LIN {X 0,Y 262.97,Z 575.386,A -85,B 0,C 180,E1 -19356.909,E2 -19356.909} C_VEL
LIN {X 0,Y 260.228,Z 588.208,A -85,B 0,C 180,E1 -19358.543,E2 -19358.543} C_VEL
LIN {X 0,Y 257.272,Z 600.423,A -85,B 0,C 180,E1 -19360.441,E2 -19360.441} C_VEL
LIN {X 0,Y 253.997,Z 612.742,A -85,B 0,C 180,E1 -19362.789,E2 -19362.789} C_VEL
LIN {X 0,Y 250.762,Z 624.067,A -85,B 0,C 180,E1 -19365.442,E2 -19365.442} C_VEL
LIN {X 0,Y 248,Z 633.546,A -85,B 0,C 180,E1 -19368.164,E2 -19368.164} C_VEL
LIN {X 0,Y 245.68,Z 641.534,A -85,B 0,C 180,E1 -19370.952,E2 -19370.952} C_VEL
LIN {X 0,Y 243.839,Z 648.227,A -85,B 0,C 180,E1 -19373.798,E2 -19373.798} C_VEL
LIN {X 0,Y 242.309,Z 653.952,A -85,B 0,C 180,E1 -19376.827,E2 -19376.827} C_VEL
LIN {X 0,Y 241.294,Z 658.236,A -85,B 0,C 180,E1 -19379.68,E2 -19379.68} C_VEL
LIN {X 0,Y 240.647,Z 661.145,A -85,B 0,C 180,E1 -19382.119,E2 -19382.119} C_VEL
LIN {X 0,Y 239.931,Z 664.333,A -85,B 0,C 180,E1 -19385.862,E2 -19385.862} C_VEL
LIN {X 0,Y 239.747,Z 665.513,A -85,B 0,C 180,E1 -19387.996,E2 -19387.996} C_VEL
LIN {X 0,Y 239.749,Z 666.237,A -85,B 0,C 180,E1 -19390.343,E2 -19390.343} C_VEL
LIN {X 0,Y 239.913,Z 666.406,A -85,B 0,C 180,E1 -19392.915,E2 -19392.915} C_VEL
LIN {X 0,Y 240.248,Z 665.992,A -85,B 0,C 180,E1 -19395.405,E2 -19395.405} C_VEL
LIN {X 0,Y 241.228,Z 664.102,A -85,B 0,C 180,E1 -19399.244,E2 -19399.244} C_VEL
LIN {X 0,Y 242.501,Z 661.254,A -85,B 0,C 180,E1 -19402.51,E2 -19402.51} C_VEL
LIN {X 0,Y 244.221,Z 657.411,A -85,B 0,C 180,E1 -19405.652,E2 -19405.652} C_VEL
LIN {X 0,Y 246.913,Z 651.612,A -85,B 0,C 180,E1 -19409.179,E2 -19409.179} C_VEL
LIN {X 0,Y 250.029,Z 644.776,A -85,B 0,C 180,E1 -19412.367,E2 -19412.367} C_VEL
LIN {X 0,Y 253.779,Z 636.355,A -85,B 0,C 180,E1 -19415.455,E2 -19415.455} C_VEL
LIN {X 0,Y 257.848,Z 626.845,A -85,B 0,C 180,E1 -19418.248,E2 -19418.248} C_VEL
LIN {X 0,Y 261.578,Z 617.491,A -85,B 0,C 180,E1 -19420.493,E2 -19420.493} C_VEL
LIN {X 0,Y 265.656,Z 606.455,A -85,B 0,C 180,E1 -19422.67,E2 -19422.67} C_VEL
LIN {X 0,Y 269.706,Z 594.368,A -85,B 0,C 180,E1 -19424.61,E2 -19424.61} C_VEL
LIN {X 0,Y 272.359,Z 585.531,A -85,B 0,C 180,E1 -19425.809,E2 -19425.809} C_VEL
LIN {X 0,Y 272.47,Z 583.373,A -85,B 0,C 180,E1 -19426.196,E2 -19426.196} C_VEL
LIN {X 0,Y 270.942,Z 574.805,A -85,B 0,C 180,E1 -19428.023,E2 -19428.023} C_VEL
LIN {X 0,Y 268.039,Z 563.986,A -85,B 0,C 180,E1 -19430.46,E2 -19430.46} C_VEL
LIN {X 0,Y 264.172,Z 554.325,A -85,B 0,C 180,E1 -19432.894,E2 -19432.894} C_VEL
LIN {X 0,Y 260.406,Z 546.743,A -85,B 0,C 180,E1 -19435.059,E2 -19435.059} C_VEL
LIN {X 0,Y 257.562,Z 542.282,A -85,B 0,C 180,E1 -19436.621,E2 -19436.621} C_VEL
LIN {X 0,Y 255.07,Z 538.329,A -85,B 0,C 180,E1 -19438.026,E2 -19438.026} C_VEL
LIN {X 0,Y 252.392,Z 534.455,A -85,B 0,C 180,E1 -19439.597,E2 -19439.597} C_VEL
LIN {X 0,Y 251.603,Z 532.992,A -85,B 0,C 180,E1 -19440.11,E2 -19440.11} C_VEL
LIN {X 0,Y 249.06,Z 530.463,A -85,B 0,C 180,E1 -19441.616,E2 -19441.616} C_VEL
LIN {X 0,Y 247.762,Z 528.054,A -85,B 0,C 180,E1 -19442.54,E2 -19442.54} C_VEL
LIN {X 0,Y 244.664,Z 526.005,A -85,B 0,C 180,E1 -19444.53,E2 -19444.53} C_VEL
LIN {X 0,Y 243.293,Z 523.765,A -85,B 0,C 180,E1 -19445.698,E2 -19445.698} C_VEL
LIN {X 0,Y 243.002,Z 522.69,A -85,B 0,C 180,E1 -19446.069,E2 -19446.069} C_VEL
LIN {X 0,Y 243.031,Z 522.727,A -85,B 0,C 180,E1 -19449.991,E2 -19449.991} C_VEL
LIN {X 0,Y 242.931,Z 523.303,A -85,B 0,C 180,E1 -19455.091,E2 -19455.091} C_VEL
LIN {X 0,Y 242.977,Z 524.161,A -85,B 0,C 180,E1 -19459.142,E2 -19459.142} C_VEL
LIN {X 0,Y 243.11,Z 525.075,A -85,B 0,C 180,E1 -19462.32,E2 -19462.32} C_VEL
LIN {X 0,Y 243.39,Z 526.569,A -85,B 0,C 180,E1 -19466.3,E2 -19466.3} C_VEL
LIN {X 0,Y 243.223,Z 527.205,A -85,B 0,C 180,E1 -19467.212,E2 -19467.212} C_VEL
LIN {X 0,Y 241.941,Z 529.538,A -85,B 0,C 180,E1 -19468.969,E2 -19468.969} C_VEL
LIN {X 0,Y 240.107,Z 534.806,A -85,B 0,C 180,E1 -19471.983,E2 -19471.983} C_VEL
LIN {X 0,Y 240.927,Z 536.647,A -85,B 0,C 180,E1 -19473.294,E2 -19473.294} C_VEL
LIN {X 0,Y 241.911,Z 537.613,A -85,B 0,C 180,E1 -19474.066,E2 -19474.066} C_VEL
LIN {X 0,Y 243.456,Z 541.241,A -85,B 0,C 180,E1 -19475.456,E2 -19475.456} C_VEL
LIN {X 0,Y 246.202,Z 544.885,A -85,B 0,C 180,E1 -19477.383,E2 -19477.383} C_VEL
LIN {X 0,Y 247.899,Z 548.7,A -85,B 0,C 180,E1 -19478.651,E2 -19478.651} C_VEL
LIN {X 0,Y 249.696,Z 551.295,A -85,B 0,C 180,E1 -19479.75,E2 -19479.75} C_VEL
LIN {X 0,Y 251.774,Z 555.814,A -85,B 0,C 180,E1 -19481.168,E2 -19481.168} C_VEL
LIN {X 0,Y 252.748,Z 557.67,A -85,B 0,C 180,E1 -19481.75,E2 -19481.75} C_VEL
LIN {X 0,Y 254.725,Z 561.939,A -85,B 0,C 180,E1 -19483.004,E2 -19483.004} C_VEL
LIN {X 0,Y 257.009,Z 569.051,A -85,B 0,C 180,E1 -19484.685,E2 -19484.685} C_VEL
LIN {X 0,Y 259.21,Z 578.738,A -85,B 0,C 180,E1 -19486.695,E2 -19486.695} C_VEL
LIN {X 0,Y 260.8,Z 588.921,A -85,B 0,C 180,E1 -19488.655,E2 -19488.655} C_VEL
LIN {X 0,Y 261.444,Z 600.468,A -85,B 0,C 180,E1 -19490.766,E2 -19490.766} C_VEL
LIN {X 0,Y 261.212,Z 611.698,A -85,B 0,C 180,E1 -19492.793,E2 -19492.793} C_VEL
LIN {X 0,Y 260.405,Z 619.56,A -85,B 0,C 180,E1 -19494.256,E2 -19494.256} C_VEL
LIN {X 0,Y 256.112,Z 631.595,A -85,B 0,C 180,E1 -19496.242,E2 -19496.242} C_VEL
LIN {X 0,Y 251.789,Z 642.638,A -85,B 0,C 180,E1 -19498.442,E2 -19498.442} C_VEL
LIN {X 0,Y 247.254,Z 653.496,A -85,B 0,C 180,E1 -19501.104,E2 -19501.104} C_VEL
LIN {X 0,Y 243.504,Z 662.394,A -85,B 0,C 180,E1 -19503.806,E2 -19503.806} C_VEL
LIN {X 0,Y 240.232,Z 670.29,A -85,B 0,C 180,E1 -19506.737,E2 -19506.737} C_VEL
LIN {X 0,Y 237.315,Z 677.59,A -85,B 0,C 180,E1 -19510.088,E2 -19510.088} C_VEL
LIN {X 0,Y 235.092,Z 683.518,A -85,B 0,C 180,E1 -19513.553,E2 -19513.553} C_VEL
LIN {X 0,Y 234.041,Z 687.003,A -85,B 0,C 180,E1 -19516.099,E2 -19516.099} C_VEL
LIN {X 0,Y 233.12,Z 690.607,A -85,B 0,C 180,E1 -19519.578,E2 -19519.578} C_VEL
LIN {X 0,Y 232.871,Z 693.033,A -85,B 0,C 180,E1 -19523.066,E2 -19523.066} C_VEL
LIN {X 0,Y 232.938,Z 694.303,A -85,B 0,C 180,E1 -19526.54,E2 -19526.54} C_VEL
LIN {X 0,Y 233.106,Z 694.406,A -85,B 0,C 180,E1 -19529.999,E2 -19529.999} C_VEL
LIN {X 0,Y 233.01,Z 693.243,A -85,B 0,C 180,E1 -19533.457,E2 -19533.457} C_VEL
LIN {X 0,Y 233.026,Z 691.945,A -85,B 0,C 180,E1 -19535.58,E2 -19535.58} C_VEL
LIN {X 0,Y 233.094,Z 688.21,A -85,B 0,C 180,E1 -19539.544,E2 -19539.544} C_VEL
LIN {X 0,Y 233.729,Z 683.513,A -85,B 0,C 180,E1 -19543.032,E2 -19543.032} C_VEL
LIN {X 0,Y 234.925,Z 677.626,A -85,B 0,C 180,E1 -19546.359,E2 -19546.359} C_VEL
LIN {X 0,Y 236.712,Z 670.612,A -85,B 0,C 180,E1 -19549.511,E2 -19549.511} C_VEL
LIN {X 0,Y 239.023,Z 662.501,A -85,B 0,C 180,E1 -19552.471,E2 -19552.471} C_VEL
LIN {X 0,Y 241.896,Z 652.756,A -85,B 0,C 180,E1 -19555.374,E2 -19555.374} C_VEL
LIN {X 0,Y 244.744,Z 642.794,A -85,B 0,C 180,E1 -19557.814,E2 -19557.814} C_VEL
LIN {X 0,Y 248.126,Z 631.005,A -85,B 0,C 180,E1 -19560.181,E2 -19560.181} C_VEL
LIN {X 0,Y 251.301,Z 619.334,A -85,B 0,C 180,E1 -19562.096,E2 -19562.096} C_VEL
LIN {X 0,Y 252.22,Z 615.752,A -85,B 0,C 180,E1 -19562.622,E2 -19562.622} C_VEL
LIN {X 0,Y 252.245,Z 609.63,A -85,B 0,C 180,E1 -19563.595,E2 -19563.595} C_VEL
LIN {X 0,Y 251.323,Z 597.034,A -85,B 0,C 180,E1 -19565.49,E2 -19565.49} C_VEL
LIN {X 0,Y 249.511,Z 583.538,A -85,B 0,C 180,E1 -19567.341,E2 -19567.341} C_VEL
LIN {X 0,Y 246.829,Z 569.413,A -85,B 0,C 180,E1 -19569.11,E2 -19569.11} C_VEL
LIN {X 0,Y 243.114,Z 554.934,A -85,B 0,C 180,E1 -19570.776,E2 -19570.776} C_VEL
LIN {X 0,Y 238.76,Z 541.769,A -85,B 0,C 180,E1 -19572.228,E2 -19572.228} C_VEL
LIN {X 0,Y 237.734,Z 538.235,A -85,B 0,C 180,E1 -19572.574,E2 -19572.574} C_VEL
LIN {X 0,Y 237.777,Z 535.861,A -85,B 0,C 180,E1 -19574.817,E2 -19574.817} C_VEL
LIN {X 0,Y 237.287,Z 532.906,A -85,B 0,C 180,E1 -19577.768,E2 -19577.768} C_VEL
LIN {X 0,Y 236.558,Z 529.52,A -85,B 0,C 180,E1 -19581.399,E2 -19581.399} C_VEL
LIN {X 0,Y 235.911,Z 525.797,A -85,B 0,C 180,E1 -19585.527,E2 -19585.527} C_VEL
LIN {X 0,Y 235.357,Z 522.081,A -85,B 0,C 180,E1 -19589.99,E2 -19589.99} C_VEL
LIN {X 0,Y 235.001,Z 519.837,A -85,B 0,C 180,E1 -19593.107,E2 -19593.107} C_VEL
LIN {X 0,Y 234.97,Z 519.844,A -85,B 0,C 180,E1 -19598,E2 -19598} C_VEL
LIN {X 0,Y 235.089,Z 519.827,A -85,B 0,C 180,E1 -19603.06,E2 -19603.06} C_VEL
LIN {X 0,Y 235.139,Z 519.815,A -85,B 0,C 180,E1 -19607.924,E2 -19607.924} C_VEL
LIN {X 0,Y 235.369,Z 519.771,A -85,B 0,C 180,E1 -19611.414,E2 -19611.414} C_VEL
LIN {X 0,Y 235.397,Z 519.778,A -85,B 0,C 180,E1 -19613.142,E2 -19613.142} C_VEL
LIN {X 0,Y 235.592,Z 519.755,A -85,B 0,C 180,E1 -19618.291,E2 -19618.291} C_VEL
LIN {X 0,Y 235.59,Z 519.741,A -85,B 0,C 180,E1 -19621.71,E2 -19621.71} C_VEL
LIN {X 0,Y 235.387,Z 519.788,A -85,B 0,C 180,E1 -19626.86,E2 -19626.86} C_VEL
LIN {X 0,Y 235.208,Z 519.795,A -85,B 0,C 180,E1 -19630.329,E2 -19630.329} C_VEL
LIN {X 0,Y 235.106,Z 519.816,A -85,B 0,C 180,E1 -19635.608,E2 -19635.608} C_VEL
LIN {X 0,Y 235.003,Z 519.837,A -85,B 0,C 180,E1 -19639.207,E2 -19639.207} C_VEL
LIN {X 0,Y 234.956,Z 519.819,A -85,B 0,C 180,E1 -19642.884,E2 -19642.884} C_VEL
LIN {X 0,Y 234.965,Z 519.83,A -85,B 0,C 180,E1 -19646.659,E2 -19646.659} C_VEL
LIN {X 0,Y 234.928,Z 519.844,A -85,B 0,C 180,E1 -19650.569,E2 -19650.569} C_VEL
LIN {X 0,Y 234.957,Z 519.821,A -85,B 0,C 180,E1 -19654.634,E2 -19654.634} C_VEL
LIN {X 0,Y 234.964,Z 519.835,A -85,B 0,C 180,E1 -19658.954,E2 -19658.954} C_VEL
LIN {X 0,Y 234.995,Z 519.832,A -85,B 0,C 180,E1 -19663.462,E2 -19663.462} C_VEL
LIN {X 0,Y 234.991,Z 519.817,A -85,B 0,C 180,E1 -19666.54,E2 -19666.54} C_VEL
LIN {X 0,Y 234.954,Z 519.846,A -85,B 0,C 180,E1 -19671.088,E2 -19671.088} C_VEL
LIN {X 0,Y 234.961,Z 519.828,A -85,B 0,C 180,E1 -19675.369,E2 -19675.369} C_VEL
LIN {X 0,Y 234.97,Z 519.844,A -85,B 0,C 180,E1 -19680.159,E2 -19680.159} C_VEL
LIN {X 0,Y 234.996,Z 519.826,A -85,B 0,C 180,E1 -19683.795,E2 -19683.795} C_VEL
LIN {X 0,Y 235.014,Z 519.831,A -85,B 0,C 180,E1 -19688.971,E2 -19688.971} C_VEL
LIN {X 0,Y 235.1,Z 519.825,A -85,B 0,C 180,E1 -19693.061,E2 -19693.061} C_VEL
LIN {X 0,Y 235.147,Z 519.821,A -85,B 0,C 180,E1 -19697.925,E2 -19697.925} C_VEL
LIN {X 0,Y 235.33,Z 519.792,A -85,B 0,C 180,E1 -19701.413,E2 -19701.413} C_VEL
LIN {X 0,Y 235.373,Z 519.791,A -85,B 0,C 180,E1 -19703.141,E2 -19703.141} C_VEL
LIN {X 0,Y 235.421,Z 519.781,A -85,B 0,C 180,E1 -19707.381,E2 -19707.381} C_VEL
LIN {X 0,Y 236.515,Z 522.659,A -85,B 0,C 180,E1 -19707.742,E2 -19707.742} C_VEL
LIN {X 0,Y 238.065,Z 524.891,A -85,B 0,C 180,E1 -19708.151,E2 -19708.151} C_VEL
LIN {X 0,Y 242.678,Z 533.731,A -85,B 0,C 180,E1 -19709.542,E2 -19709.542} C_VEL
LIN {X 0,Y 249.035,Z 548.124,A -85,B 0,C 180,E1 -19711.775,E2 -19711.775} C_VEL
LIN {X 0,Y 252.052,Z 557.462,A -85,B 0,C 180,E1 -19713.198,E2 -19713.198} C_VEL
LIN {X 0,Y 255.332,Z 570.437,A -85,B 0,C 180,E1 -19715.255,E2 -19715.255} C_VEL
LIN {X 0,Y 256.488,Z 576.766,A -85,B 0,C 180,E1 -19716.293,E2 -19716.293} C_VEL
LIN {X 0,Y 253.332,Z 590.847,A -85,B 0,C 180,E1 -19718.175,E2 -19718.175} C_VEL
LIN {X 0,Y 250.031,Z 603.805,A -85,B 0,C 180,E1 -19720.324,E2 -19720.324} C_VEL
LIN {X 0,Y 246.656,Z 615.754,A -85,B 0,C 180,E1 -19722.758,E2 -19722.758} C_VEL
LIN {X 0,Y 243.418,Z 626.66,A -85,B 0,C 180,E1 -19725.49,E2 -19725.49} C_VEL
LIN {X 0,Y 240.665,Z 635.779,A -85,B 0,C 180,E1 -19728.297,E2 -19728.297} C_VEL
LIN {X 0,Y 238.341,Z 643.461,A -85,B 0,C 180,E1 -19731.175,E2 -19731.175} C_VEL
LIN {X 0,Y 236.222,Z 650.859,A -85,B 0,C 180,E1 -19734.616,E2 -19734.616} C_VEL
LIN {X 0,Y 234.883,Z 655.996,A -85,B 0,C 180,E1 -19737.632,E2 -19737.632} C_VEL
LIN {X 0,Y 233.887,Z 660.153,A -85,B 0,C 180,E1 -19740.719,E2 -19740.719} C_VEL
LIN {X 0,Y 233.36,Z 662.351,A -85,B 0,C 180,E1 -19742.827,E2 -19742.827} C_VEL
LIN {X 0,Y 232.882,Z 664.441,A -85,B 0,C 180,E1 -19745.429,E2 -19745.429} C_VEL
LIN {X 0,Y 232.633,Z 666.379,A -85,B 0,C 180,E1 -19749.378,E2 -19749.378} C_VEL
LIN {X 0,Y 232.725,Z 666.833,A -85,B 0,C 180,E1 -19751.634,E2 -19751.634} C_VEL
LIN {X 0,Y 232.936,Z 666.819,A -85,B 0,C 180,E1 -19753.943,E2 -19753.943} C_VEL
LIN {X 0,Y 233.325,Z 666.251,A -85,B 0,C 180,E1 -19756.295,E2 -19756.295} C_VEL
LIN {X 0,Y 233.963,Z 665.147,A -85,B 0,C 180,E1 -19758.675,E2 -19758.675} C_VEL
LIN {X 0,Y 235.285,Z 662.487,A -85,B 0,C 180,E1 -19762.261,E2 -19762.261} C_VEL
LIN {X 0,Y 237.336,Z 658.263,A -85,B 0,C 180,E1 -19766.01,E2 -19766.01} C_VEL
LIN {X 0,Y 239.932,Z 653.095,A -85,B 0,C 180,E1 -19769.35,E2 -19769.35} C_VEL
LIN {X 0,Y 242.909,Z 647.003,A -85,B 0,C 180,E1 -19772.423,E2 -19772.423} C_VEL
LIN {X 0,Y 246.185,Z 640.109,A -85,B 0,C 180,E1 -19775.203,E2 -19775.203} C_VEL
LIN {X 0,Y 250.414,Z 630.965,A -85,B 0,C 180,E1 -19778.172,E2 -19778.172} C_VEL
LIN {X 0,Y 254.916,Z 620.513,A -85,B 0,C 180,E1 -19780.889,E2 -19780.889} C_VEL
LIN {X 0,Y 259.401,Z 609.166,A -85,B 0,C 180,E1 -19783.269,E2 -19783.269} C_VEL
LIN {X 0,Y 263.785,Z 596.954,A -85,B 0,C 180,E1 -19785.338,E2 -19785.338} C_VEL
LIN {X 0,Y 266.902,Z 587.098,A -85,B 0,C 180,E1 -19786.717,E2 -19786.717} C_VEL
LIN {X 0,Y 265.723,Z 578.921,A -85,B 0,C 180,E1 -19788.558,E2 -19788.558} C_VEL
LIN {X 0,Y 263.505,Z 569.481,A -85,B 0,C 180,E1 -19790.791,E2 -19790.791} C_VEL
LIN {X 0,Y 260.847,Z 561.758,A -85,B 0,C 180,E1 -19792.803,E2 -19792.803} C_VEL
LIN {X 0,Y 257.119,Z 553.218,A -85,B 0,C 180,E1 -19795.296,E2 -19795.296} C_VEL
LIN {X 0,Y 254.632,Z 548.771,A -85,B 0,C 180,E1 -19796.835,E2 -19796.835} C_VEL
LIN {X 0,Y 251.808,Z 544.068,A -85,B 0,C 180,E1 -19798.63,E2 -19798.63} C_VEL
LIN {X 0,Y 249.334,Z 540.251,A -85,B 0,C 180,E1 -19800.226,E2 -19800.226} C_VEL
LIN {X 0,Y 248.552,Z 539.039,A -85,B 0,C 180,E1 -19800.759,E2 -19800.759} C_VEL
LIN {X 0,Y 246.294,Z 536.366,A -85,B 0,C 180,E1 -19802.277,E2 -19802.277} C_VEL
LIN {X 0,Y 245.257,Z 534.562,A -85,B 0,C 180,E1 -19803.079,E2 -19803.079} C_VEL
LIN {X 0,Y 242.481,Z 532.36,A -85,B 0,C 180,E1 -19805.092,E2 -19805.092} C_VEL
LIN {X 0,Y 241.054,Z 529.742,A -85,B 0,C 180,E1 -19806.434,E2 -19806.434} C_VEL
LIN {X 0,Y 237.552,Z 527.249,A -85,B 0,C 180,E1 -19809.794,E2 -19809.794} C_VEL
LIN {X 0,Y 236.193,Z 525.11,A -85,B 0,C 180,E1 -19811.804,E2 -19811.804} C_VEL
LIN {X 0,Y 235.995,Z 524.537,A -85,B 0,C 180,E1 -19812.25,E2 -19812.25} C_VEL
LIN {X 0,Y 236.03,Z 524.997,A -85,B 0,C 180,E1 -19815.544,E2 -19815.544} C_VEL
LIN {X 0,Y 236.063,Z 525.768,A -85,B 0,C 180,E1 -19819.116,E2 -19819.116} C_VEL
LIN {X 0,Y 236.222,Z 526.838,A -85,B 0,C 180,E1 -19822.753,E2 -19822.753} C_VEL
LIN {X 0,Y 236.505,Z 528.439,A -85,B 0,C 180,E1 -19826.94,E2 -19826.94} C_VEL
LIN {X 0,Y 236.652,Z 529.379,A -85,B 0,C 180,E1 -19828.611,E2 -19828.611} C_VEL
LIN {X 0,Y 238.401,Z 533.574,A -85,B 0,C 180,E1 -19830.95,E2 -19830.95} C_VEL
LIN {X 0,Y 240.927,Z 536.647,A -85,B 0,C 180,E1 -19833.294,E2 -19833.294} C_VEL
LIN {X 0,Y 241.916,Z 538.055,A -85,B 0,C 180,E1 -19834.124,E2 -19834.124} C_VEL
LIN {X 0,Y 243.061,Z 541.33,A -85,B 0,C 180,E1 -19835.247,E2 -19835.247} C_VEL
LIN {X 0,Y 243.881,Z 545.39,A -85,B 0,C 180,E1 -19836.251,E2 -19836.251} C_VEL
LIN {X 0,Y 245.389,Z 554.106,A -85,B 0,C 180,E1 -19838.231,E2 -19838.231} C_VEL
LIN {X 0,Y 246.185,Z 556.608,A -85,B 0,C 180,E1 -19838.953,E2 -19838.953} C_VEL
LIN {X 0,Y 248.839,Z 562.367,A -85,B 0,C 180,E1 -19840.919,E2 -19840.919} C_VEL
LIN {X 0,Y 251.791,Z 570.132,A -85,B 0,C 180,E1 -19843.145,E2 -19843.145} C_VEL
LIN {X 0,Y 253.95,Z 580.016,A -85,B 0,C 180,E1 -19845.372,E2 -19845.372} C_VEL
LIN {X 0,Y 255.419,Z 590.889,A -85,B 0,C 180,E1 -19847.614,E2 -19847.614} C_VEL
LIN {X 0,Y 255.913,Z 601.984,A -85,B 0,C 180,E1 -19849.761,E2 -19849.761} C_VEL
LIN {X 0,Y 255.478,Z 612.786,A -85,B 0,C 180,E1 -19851.841,E2 -19851.841} C_VEL
LIN {X 0,Y 254.531,Z 620.794,A -85,B 0,C 180,E1 -19853.393,E2 -19853.393} C_VEL
LIN {X 0,Y 250.259,Z 632.18,A -85,B 0,C 180,E1 -19855.342,E2 -19855.342} C_VEL
LIN {X 0,Y 245.782,Z 643.009,A -85,B 0,C 180,E1 -19857.578,E2 -19857.578} C_VEL
LIN {X 0,Y 241.047,Z 653.694,A -85,B 0,C 180,E1 -19860.287,E2 -19860.287} C_VEL
LIN {X 0,Y 237.004,Z 662.754,A -85,B 0,C 180,E1 -19863.121,E2 -19863.121} C_VEL
LIN {X 0,Y 233.671,Z 670.313,A -85,B 0,C 180,E1 -19866.044,E2 -19866.044} C_VEL
LIN {X 0,Y 230.591,Z 677.488,A -85,B 0,C 180,E1 -19869.482,E2 -19869.482} C_VEL
LIN {X 0,Y 228.152,Z 683.517,A -85,B 0,C 180,E1 -19873.164,E2 -19873.164} C_VEL
LIN {X 0,Y 227.085,Z 686.778,A -85,B 0,C 180,E1 -19875.664,E2 -19875.664} C_VEL
LIN {X 0,Y 226.08,Z 690.314,A -85,B 0,C 180,E1 -19879.25,E2 -19879.25} C_VEL
LIN {X 0,Y 225.785,Z 692.672,A -85,B 0,C 180,E1 -19882.847,E2 -19882.847} C_VEL
LIN {X 0,Y 225.855,Z 693.883,A -85,B 0,C 180,E1 -19886.431,E2 -19886.431} C_VEL
LIN {X 0,Y 226.027,Z 693.927,A -85,B 0,C 180,E1 -19889.999,E2 -19889.999} C_VEL
LIN {X 0,Y 225.924,Z 692.734,A -85,B 0,C 180,E1 -19893.566,E2 -19893.566} C_VEL
LIN {X 0,Y 225.955,Z 691.531,A -85,B 0,C 180,E1 -19895.554,E2 -19895.554} C_VEL
LIN {X 0,Y 225.948,Z 688.536,A -85,B 0,C 180,E1 -19898.946,E2 -19898.946} C_VEL
LIN {X 0,Y 226.476,Z 684.098,A -85,B 0,C 180,E1 -19902.545,E2 -19902.545} C_VEL
LIN {X 0,Y 227.696,Z 678.236,A -85,B 0,C 180,E1 -19906.127,E2 -19906.127} C_VEL
LIN {X 0,Y 229.626,Z 670.797,A -85,B 0,C 180,E1 -19909.673,E2 -19909.673} C_VEL
LIN {X 0,Y 231.999,Z 662.821,A -85,B 0,C 180,E1 -19912.719,E2 -19912.719} C_VEL
LIN {X 0,Y 234.956,Z 653.23,A -85,B 0,C 180,E1 -19915.703,E2 -19915.703} C_VEL
LIN {X 0,Y 237.827,Z 643.434,A -85,B 0,C 180,E1 -19918.216,E2 -19918.216} C_VEL
LIN {X 0,Y 241.331,Z 631.861,A -85,B 0,C 180,E1 -19920.638,E2 -19920.638} C_VEL
LIN {X 0,Y 244.186,Z 621.693,A -85,B 0,C 180,E1 -19922.414,E2 -19922.414} C_VEL
LIN {X 0,Y 245.773,Z 615.207,A -85,B 0,C 180,E1 -19923.407,E2 -19923.407} C_VEL
LIN {X 0,Y 245.147,Z 602.047,A -85,B 0,C 180,E1 -19925.56,E2 -19925.56} C_VEL
LIN {X 0,Y 243.766,Z 589.315,A -85,B 0,C 180,E1 -19927.447,E2 -19927.447} C_VEL
LIN {X 0,Y 241.623,Z 575.898,A -85,B 0,C 180,E1 -19929.248,E2 -19929.248} C_VEL
LIN {X 0,Y 238.406,Z 561.756,A -85,B 0,C 180,E1 -19931.021,E2 -19931.021} C_VEL
LIN {X 0,Y 234.503,Z 548.503,A -85,B 0,C 180,E1 -19932.605,E2 -19932.605} C_VEL
LIN {X 0,Y 231.927,Z 541.355,A -85,B 0,C 180,E1 -19933.442,E2 -19933.442} C_VEL
LIN {X 0,Y 230.914,Z 538.378,A -85,B 0,C 180,E1 -19933.768,E2 -19933.768} C_VEL
LIN {X 0,Y 230.86,Z 537.772,A -85,B 0,C 180,E1 -19933.853,E2 -19933.853} C_VEL
LIN {X 0,Y 230.254,Z 533.886,A -85,B 0,C 180,E1 -19937.818,E2 -19937.818} C_VEL
LIN {X 0,Y 229.287,Z 529.343,A -85,B 0,C 180,E1 -19942.836,E2 -19942.836} C_VEL
LIN {X 0,Y 228.791,Z 526.237,A -85,B 0,C 180,E1 -19946.433,E2 -19946.433} C_VEL
LIN {X 0,Y 228.326,Z 522.984,A -85,B 0,C 180,E1 -19950.496,E2 -19950.496} C_VEL
LIN {X 0,Y 227.961,Z 520.716,A -85,B 0,C 180,E1 -19953.575,E2 -19953.575} C_VEL
LIN {X 0,Y 227.94,Z 520.719,A -85,B 0,C 180,E1 -19958.286,E2 -19958.286} C_VEL
LIN {X 0,Y 228.027,Z 520.706,A -85,B 0,C 180,E1 -19962.826,E2 -19962.826} C_VEL
LIN {X 0,Y 228.087,Z 520.696,A -85,B 0,C 180,E1 -19967.545,E2 -19967.545} C_VEL
LIN {X 0,Y 228.298,Z 520.649,A -85,B 0,C 180,E1 -19971.146,E2 -19971.146} C_VEL
LIN {X 0,Y 228.348,Z 520.655,A -85,B 0,C 180,E1 -19972.929,E2 -19972.929} C_VEL
LIN {X 0,Y 228.55,Z 520.631,A -85,B 0,C 180,E1 -19978.239,E2 -19978.239} C_VEL
LIN {X 0,Y 228.549,Z 520.616,A -85,B 0,C 180,E1 -19981.763,E2 -19981.763} C_VEL
LIN {X 0,Y 228.334,Z 520.668,A -85,B 0,C 180,E1 -19987.073,E2 -19987.073} C_VEL
LIN {X 0,Y 228.139,Z 520.672,A -85,B 0,C 180,E1 -19990.652,E2 -19990.652} C_VEL
LIN {X 0,Y 228.056,Z 520.685,A -85,B 0,C 180,E1 -19994.273,E2 -19994.273} C_VEL
LIN {X 0,Y 227.998,Z 520.709,A -85,B 0,C 180,E1 -19997.955,E2 -19997.955} C_VEL
LIN {X 0,Y 227.925,Z 520.699,A -85,B 0,C 180,E1 -20002.33,E2 -20002.33} C_VEL
LIN {X 0,Y 227.938,Z 520.705,A -85,B 0,C 180,E1 -20006.604,E2 -20006.604} C_VEL
LIN {X 0,Y 227.904,Z 520.72,A -85,B 0,C 180,E1 -20010.297,E2 -20010.297} C_VEL
LIN {X 0,Y 227.886,Z 520.705,A -85,B 0,C 180,E1 -20013.72,E2 -20013.72} C_VEL
LIN {X 0,Y 227.869,Z 520.714,A -85,B 0,C 180,E1 -20018.087,E2 -20018.087} C_VEL
LIN {X 0,Y 227.932,Z 520.715,A -85,B 0,C 180,E1 -20022.715,E2 -20022.715} C_VEL
LIN {X 0,Y 227.925,Z 520.7,A -85,B 0,C 180,E1 -20027.286,E2 -20027.286} C_VEL
LIN {X 0,Y 227.871,Z 520.727,A -85,B 0,C 180,E1 -20031.916,E2 -20031.916} C_VEL
LIN {X 0,Y 227.891,Z 520.71,A -85,B 0,C 180,E1 -20036.375,E2 -20036.375} C_VEL
LIN {X 0,Y 227.92,Z 520.722,A -85,B 0,C 180,E1 -20040.44,E2 -20040.44} C_VEL
LIN {X 0,Y 227.931,Z 520.708,A -85,B 0,C 180,E1 -20044.428,E2 -20044.428} C_VEL
LIN {X 0,Y 227.965,Z 520.711,A -85,B 0,C 180,E1 -20048.289,E2 -20048.289} C_VEL
LIN {X 0,Y 228.038,Z 520.704,A -85,B 0,C 180,E1 -20052.827,E2 -20052.827} C_VEL
LIN {X 0,Y 228.095,Z 520.697,A -85,B 0,C 180,E1 -20057.546,E2 -20057.546} C_VEL
LIN {X 0,Y 228.267,Z 520.67,A -85,B 0,C 180,E1 -20061.146,E2 -20061.146} C_VEL
LIN {X 0,Y 228.323,Z 520.67,A -85,B 0,C 180,E1 -20062.929,E2 -20062.929} C_VEL
LIN {X 0,Y 228.251,Z 520.679,A -85,B 0,C 180,E1 -20066.084,E2 -20066.084} C_VEL
LIN {X 0,Y 229.317,Z 523.568,A -85,B 0,C 180,E1 -20066.487,E2 -20066.487} C_VEL
LIN {X 0,Y 230.971,Z 525.981,A -85,B 0,C 180,E1 -20066.954,E2 -20066.954} C_VEL
LIN {X 0,Y 235.225,Z 533.304,A -85,B 0,C 180,E1 -20068.23,E2 -20068.23} C_VEL
LIN {X 0,Y 240.128,Z 544.236,A -85,B 0,C 180,E1 -20070.001,E2 -20070.001} C_VEL
LIN {X 0,Y 244.225,Z 554.06,A -85,B 0,C 180,E1 -20071.65,E2 -20071.65} C_VEL
LIN {X 0,Y 247.847,Z 567.534,A -85,B 0,C 180,E1 -20073.812,E2 -20073.812} C_VEL
LIN {X 0,Y 250.012,Z 578.067,A -85,B 0,C 180,E1 -20075.631,E2 -20075.631} C_VEL
LIN {X 0,Y 246.898,Z 591.679,A -85,B 0,C 180,E1 -20077.515,E2 -20077.515} C_VEL
LIN {X 0,Y 243.749,Z 603.654,A -85,B 0,C 180,E1 -20079.544,E2 -20079.544} C_VEL
LIN {X 0,Y 240.222,Z 615.707,A -85,B 0,C 180,E1 -20082.032,E2 -20082.032} C_VEL
LIN {X 0,Y 237.105,Z 625.839,A -85,B 0,C 180,E1 -20084.593,E2 -20084.593} C_VEL
LIN {X 0,Y 234.179,Z 635.167,A -85,B 0,C 180,E1 -20087.465,E2 -20087.465} C_VEL
LIN {X 0,Y 231.516,Z 643.647,A -85,B 0,C 180,E1 -20090.675,E2 -20090.675} C_VEL
LIN {X 0,Y 229.788,Z 649.613,A -85,B 0,C 180,E1 -20093.429,E2 -20093.429} C_VEL
LIN {X 0,Y 228.129,Z 655.356,A -85,B 0,C 180,E1 -20096.693,E2 -20096.693} C_VEL
LIN {X 0,Y 227.014,Z 659.736,A -85,B 0,C 180,E1 -20099.905,E2 -20099.905} C_VEL
LIN {X 0,Y 226.23,Z 662.963,A -85,B 0,C 180,E1 -20102.988,E2 -20102.988} C_VEL
LIN {X 0,Y 225.705,Z 665.42,A -85,B 0,C 180,E1 -20106.273,E2 -20106.273} C_VEL
LIN {X 0,Y 225.544,Z 666.598,A -85,B 0,C 180,E1 -20108.829,E2 -20108.829} C_VEL
LIN {X 0,Y 225.647,Z 667.241,A -85,B 0,C 180,E1 -20111.624,E2 -20111.624} C_VEL
LIN {X 0,Y 225.903,Z 667.258,A -85,B 0,C 180,E1 -20114.311,E2 -20114.311} C_VEL
LIN {X 0,Y 226.699,Z 666.16,A -85,B 0,C 180,E1 -20118.076,E2 -20118.076} C_VEL
LIN {X 0,Y 228.06,Z 663.711,A -85,B 0,C 180,E1 -20121.95,E2 -20121.95} C_VEL
LIN {X 0,Y 229.988,Z 660.074,A -85,B 0,C 180,E1 -20125.596,E2 -20125.596} C_VEL
LIN {X 0,Y 232.543,Z 655.264,A -85,B 0,C 180,E1 -20129.083,E2 -20129.083} C_VEL
LIN {X 0,Y 235.608,Z 649.44,A -85,B 0,C 180,E1 -20132.319,E2 -20132.319} C_VEL
LIN {X 0,Y 239.349,Z 642.069,A -85,B 0,C 180,E1 -20135.54,E2 -20135.54} C_VEL
LIN {X 0,Y 243.465,Z 633.702,A -85,B 0,C 180,E1 -20138.442,E2 -20138.442} C_VEL
LIN {X 0,Y 247.847,Z 624.245,A -85,B 0,C 180,E1 -20141.108,E2 -20141.108} C_VEL
LIN {X 0,Y 252.483,Z 613.491,A -85,B 0,C 180,E1 -20143.553,E2 -20143.553} C_VEL
LIN {X 0,Y 257.092,Z 601.541,A -85,B 0,C 180,E1 -20145.757,E2 -20145.757} C_VEL
LIN {X 0,Y 261.269,Z 589.396,A -85,B 0,C 180,E1 -20147.572,E2 -20147.572} C_VEL
LIN {X 0,Y 260.226,Z 581.477,A -85,B 0,C 180,E1 -20149.478,E2 -20149.478} C_VEL
LIN {X 0,Y 258.245,Z 572.358,A -85,B 0,C 180,E1 -20151.785,E2 -20151.785} C_VEL
LIN {X 0,Y 255.493,Z 564.194,A -85,B 0,C 180,E1 -20154.091,E2 -20154.091} C_VEL
LIN {X 0,Y 252.963,Z 558.124,A -85,B 0,C 180,E1 -20156.018,E2 -20156.018} C_VEL
LIN {X 0,Y 248.426,Z 549.809,A -85,B 0,C 180,E1 -20159.199,E2 -20159.199} C_VEL
LIN {X 0,Y 246.381,Z 546.457,A -85,B 0,C 180,E1 -20160.689,E2 -20160.689} C_VEL
LIN {X 0,Y 245.553,Z 545.136,A -85,B 0,C 180,E1 -20161.332,E2 -20161.332} C_VEL
LIN {X 0,Y 243.239,Z 541.895,A -85,B 0,C 180,E1 -20163.089,E2 -20163.089} C_VEL
LIN {X 0,Y 242.755,Z 541.084,A -85,B 0,C 180,E1 -20163.5,E2 -20163.5} C_VEL
LIN {X 0,Y 240.113,Z 538.667,A -85,B 0,C 180,E1 -20165.64,E2 -20165.64} C_VEL
LIN {X 0,Y 238.87,Z 536.212,A -85,B 0,C 180,E1 -20166.97,E2 -20166.97} C_VEL
LIN {X 0,Y 235.95,Z 534.077,A -85,B 0,C 180,E1 -20170.05,E2 -20170.05} C_VEL
LIN {X 0,Y 234.621,Z 531.814,A -85,B 0,C 180,E1 -20172.213,E2 -20172.213} C_VEL
LIN {X 0,Y 234.116,Z 531.456,A -85,B 0,C 180,E1 -20173.011,E2 -20173.011} C_VEL
LIN {X 0,Y 232.115,Z 531.549,A -85,B 0,C 180,E1 -20178.536,E2 -20178.536} C_VEL
LIN {X 0,Y 232.383,Z 532.859,A -85,B 0,C 180,E1 -20182.849,E2 -20182.849} C_VEL
LIN {X 0,Y 234.972,Z 536.052,A -85,B 0,C 180,E1 -20188.104,E2 -20188.104} C_VEL
LIN {X 0,Y 236.733,Z 540.453,A -85,B 0,C 180,E1 -20190.706,E2 -20190.706} C_VEL
LIN {X 0,Y 239.621,Z 544.115,A -85,B 0,C 180,E1 -20193.527,E2 -20193.527} C_VEL
LIN {X 0,Y 241.439,Z 548.31,A -85,B 0,C 180,E1 -20195.315,E2 -20195.315} C_VEL
LIN {X 0,Y 243.355,Z 550.972,A -85,B 0,C 180,E1 -20196.763,E2 -20196.763} C_VEL
LIN {X 0,Y 245.264,Z 555.273,A -85,B 0,C 180,E1 -20198.356,E2 -20198.356} C_VEL
LIN {X 0,Y 246.185,Z 556.608,A -85,B 0,C 180,E1 -20198.953,E2 -20198.953} C_VEL
LIN {X 0,Y 247.235,Z 560.443,A -85,B 0,C 180,E1 -20199.972,E2 -20199.972} C_VEL
LIN {X 0,Y 247.772,Z 564.931,A -85,B 0,C 180,E1 -20200.872,E2 -20200.872} C_VEL
LIN {X 0,Y 248.273,Z 577.63,A -85,B 0,C 180,E1 -20203.145,E2 -20203.145} C_VEL
LIN {X 0,Y 248.681,Z 580.51,A -85,B 0,C 180,E1 -20203.784,E2 -20203.784} C_VEL
LIN {X 0,Y 250.187,Z 592.768,A -85,B 0,C 180,E1 -20206.511,E2 -20206.511} C_VEL
LIN {X 0,Y 250.478,Z 603.534,A -85,B 0,C 180,E1 -20208.727,E2 -20208.727} C_VEL
LIN {X 0,Y 249.717,Z 615.113,A -85,B 0,C 180,E1 -20211.065,E2 -20211.065} C_VEL
LIN {X 0,Y 248.403,Z 623.323,A -85,B 0,C 180,E1 -20212.723,E2 -20212.723} C_VEL
LIN {X 0,Y 243.631,Z 634.691,A -85,B 0,C 180,E1 -20214.764,E2 -20214.764} C_VEL
LIN {X 0,Y 239.078,Z 645.044,A -85,B 0,C 180,E1 -20217.055,E2 -20217.055} C_VEL
LIN {X 0,Y 234.239,Z 655.307,A -85,B 0,C 180,E1 -20219.83,E2 -20219.83} C_VEL
LIN {X 0,Y 230.122,Z 663.957,A -85,B 0,C 180,E1 -20222.735,E2 -20222.735} C_VEL
LIN {X 0,Y 227.168,Z 670.352,A -85,B 0,C 180,E1 -20225.313,E2 -20225.313} C_VEL
LIN {X 0,Y 223.876,Z 677.432,A -85,B 0,C 180,E1 -20228.837,E2 -20228.837} C_VEL
LIN {X 0,Y 221.54,Z 682.63,A -85,B 0,C 180,E1 -20232.118,E2 -20232.118} C_VEL
LIN {X 0,Y 220.112,Z 686.528,A -85,B 0,C 180,E1 -20235.2,E2 -20235.2} C_VEL
LIN {X 0,Y 219.057,Z 690.031,A -85,B 0,C 180,E1 -20238.901,E2 -20238.901} C_VEL
LIN {X 0,Y 218.687,Z 692.318,A -85,B 0,C 180,E1 -20242.613,E2 -20242.613} C_VEL
LIN {X 0,Y 218.77,Z 693.142,A -85,B 0,C 180,E1 -20244.79,E2 -20244.79} C_VEL
LIN {X 0,Y 218.862,Z 693.605,A -85,B 0,C 180,E1 -20248.159,E2 -20248.159} C_VEL
LIN {X 0,Y 218.951,Z 693.449,A -85,B 0,C 180,E1 -20249.999,E2 -20249.999} C_VEL
LIN {X 0,Y 218.842,Z 692.209,A -85,B 0,C 180,E1 -20253.682,E2 -20253.682} C_VEL
LIN {X 0,Y 218.883,Z 691.117,A -85,B 0,C 180,E1 -20255.527,E2 -20255.527} C_VEL
LIN {X 0,Y 218.895,Z 687.929,A -85,B 0,C 180,E1 -20259.237,E2 -20259.237} C_VEL
LIN {X 0,Y 219.48,Z 683.419,A -85,B 0,C 180,E1 -20262.952,E2 -20262.952} C_VEL
LIN {X 0,Y 220.788,Z 677.48,A -85,B 0,C 180,E1 -20266.646,E2 -20266.646} C_VEL
LIN {X 0,Y 222.869,Z 669.96,A -85,B 0,C 180,E1 -20270.295,E2 -20270.295} C_VEL
LIN {X 0,Y 225.381,Z 661.894,A -85,B 0,C 180,E1 -20273.426,E2 -20273.426} C_VEL
LIN {X 0,Y 228.31,Z 652.58,A -85,B 0,C 180,E1 -20276.381,E2 -20276.381} C_VEL
LIN {X 0,Y 231.522,Z 642.287,A -85,B 0,C 180,E1 -20279.056,E2 -20279.056} C_VEL
LIN {X 0,Y 235.113,Z 630.56,A -85,B 0,C 180,E1 -20281.539,E2 -20281.539} C_VEL
LIN {X 0,Y 238.506,Z 618.973,A -85,B 0,C 180,E1 -20283.537,E2 -20283.537} C_VEL
LIN {X 0,Y 239.137,Z 616.384,A -85,B 0,C 180,E1 -20283.943,E2 -20283.943} C_VEL
LIN {X 0,Y 238.675,Z 603.978,A -85,B 0,C 180,E1 -20286.078,E2 -20286.078} C_VEL
LIN {X 0,Y 237.435,Z 591.248,A -85,B 0,C 180,E1 -20288.063,E2 -20288.063} C_VEL
LIN {X 0,Y 235.446,Z 577.804,A -85,B 0,C 180,E1 -20289.976,E2 -20289.976} C_VEL
LIN {X 0,Y 232.073,Z 562.373,A -85,B 0,C 180,E1 -20292.018,E2 -20292.018} C_VEL
LIN {X 0,Y 228.051,Z 548.888,A -85,B 0,C 180,E1 -20293.713,E2 -20293.713} C_VEL
LIN {X 0,Y 225.165,Z 541.382,A -85,B 0,C 180,E1 -20294.679,E2 -20294.679} C_VEL
LIN {X 0,Y 223.772,Z 538.165,A -85,B 0,C 180,E1 -20295.117,E2 -20295.117} C_VEL
LIN {X 0,Y 223.629,Z 537.286,A -85,B 0,C 180,E1 -20295.239,E2 -20295.239} C_VEL
LIN {X 0,Y 223.043,Z 534.246,A -85,B 0,C 180,E1 -20298.571,E2 -20298.571} C_VEL
LIN {X 0,Y 222.244,Z 530.204,A -85,B 0,C 180,E1 -20303.071,E2 -20303.071} C_VEL
LIN {X 0,Y 221.649,Z 526.707,A -85,B 0,C 180,E1 -20307.383,E2 -20307.383} C_VEL
LIN {X 0,Y 221.21,Z 523.459,A -85,B 0,C 180,E1 -20311.54,E2 -20311.54} C_VEL
LIN {X 0,Y 220.883,Z 521.596,A -85,B 0,C 180,E1 -20314.31,E2 -20314.31} C_VEL
LIN {X 0,Y 220.858,Z 521.602,A -85,B 0,C 180,E1 -20317.552,E2 -20317.552} C_VEL
LIN {X 0,Y 220.977,Z 521.584,A -85,B 0,C 180,E1 -20322.571,E2 -20322.571} C_VEL
LIN {X 0,Y 221.019,Z 521.579,A -85,B 0,C 180,E1 -20327.14,E2 -20327.14} C_VEL
LIN {X 0,Y 221.229,Z 521.528,A -85,B 0,C 180,E1 -20330.861,E2 -20330.861} C_VEL
LIN {X 0,Y 221.299,Z 521.532,A -85,B 0,C 180,E1 -20332.703,E2 -20332.703} C_VEL
LIN {X 0,Y 221.508,Z 521.508,A -85,B 0,C 180,E1 -20338.183,E2 -20338.183} C_VEL
LIN {X 0,Y 221.507,Z 521.492,A -85,B 0,C 180,E1 -20341.819,E2 -20341.819} C_VEL
LIN {X 0,Y 221.266,Z 521.549,A -85,B 0,C 180,E1 -20347.3,E2 -20347.3} C_VEL
LIN {X 0,Y 221.061,Z 521.547,A -85,B 0,C 180,E1 -20350.998,E2 -20350.998} C_VEL
LIN {X 0,Y 221.01,Z 521.576,A -85,B 0,C 180,E1 -20356.631,E2 -20356.631} C_VEL
LIN {X 0,Y 220.887,Z 521.588,A -85,B 0,C 180,E1 -20360.487,E2 -20360.487} C_VEL
LIN {X 0,Y 220.862,Z 521.566,A -85,B 0,C 180,E1 -20364.436,E2 -20364.436} C_VEL
LIN {X 0,Y 220.832,Z 521.599,A -85,B 0,C 180,E1 -20368.515,E2 -20368.515} C_VEL
LIN {X 0,Y 220.821,Z 521.595,A -85,B 0,C 180,E1 -20372.756,E2 -20372.756} C_VEL
LIN {X 0,Y 220.836,Z 521.582,A -85,B 0,C 180,E1 -20377.29,E2 -20377.29} C_VEL
LIN {X 0,Y 220.872,Z 521.596,A -85,B 0,C 180,E1 -20381.93,E2 -20381.93} C_VEL
LIN {X 0,Y 220.871,Z 521.574,A -85,B 0,C 180,E1 -20385.573,E2 -20385.573} C_VEL
LIN {X 0,Y 220.856,Z 521.6,A -85,B 0,C 180,E1 -20389.794,E2 -20389.794} C_VEL
LIN {X 0,Y 220.835,Z 521.602,A -85,B 0,C 180,E1 -20392.797,E2 -20392.797} C_VEL
LIN {X 0,Y 220.825,Z 521.595,A -85,B 0,C 180,E1 -20397.247,E2 -20397.247} C_VEL
LIN {X 0,Y 220.838,Z 521.599,A -85,B 0,C 180,E1 -20401.488,E2 -20401.488} C_VEL
LIN {X 0,Y 220.871,Z 521.594,A -85,B 0,C 180,E1 -20405.567,E2 -20405.567} C_VEL
LIN {X 0,Y 220.896,Z 521.583,A -85,B 0,C 180,E1 -20409.516,E2 -20409.516} C_VEL
LIN {X 0,Y 221.02,Z 521.581,A -85,B 0,C 180,E1 -20413.372,E2 -20413.372} C_VEL
LIN {X 0,Y 221.091,Z 521.569,A -85,B 0,C 180,E1 -20419.006,E2 -20419.006} C_VEL
LIN {X 0,Y 221.259,Z 521.55,A -85,B 0,C 180,E1 -20422.702,E2 -20422.702} C_VEL
LIN {X 0,Y 221.15,Z 521.561,A -85,B 0,C 180,E1 -20424.759,E2 -20424.759} C_VEL
LIN {X 0,Y 222.043,Z 524.243,A -85,B 0,C 180,E1 -20425.098,E2 -20425.098} C_VEL
LIN {X 0,Y 223.67,Z 526.555,A -85,B 0,C 180,E1 -20425.59,E2 -20425.59} C_VEL
LIN {X 0,Y 229.862,Z 537.19,A -85,B 0,C 180,E1 -20427.589,E2 -20427.589} C_VEL
LIN {X 0,Y 234.938,Z 548.849,A -85,B 0,C 180,E1 -20429.585,E2 -20429.585} C_VEL
LIN {X 0,Y 238.295,Z 557.12,A -85,B 0,C 180,E1 -20431.069,E2 -20431.069} C_VEL
LIN {X 0,Y 241.422,Z 569.334,A -85,B 0,C 180,E1 -20433.129,E2 -20433.129} C_VEL
LIN {X 0,Y 243.558,Z 579.566,A -85,B 0,C 180,E1 -20434.967,E2 -20434.967} C_VEL
LIN {X 0,Y 240.373,Z 592.943,A -85,B 0,C 180,E1 -20436.888,E2 -20436.888} C_VEL
LIN {X 0,Y 236.816,Z 605.906,A -85,B 0,C 180,E1 -20439.179,E2 -20439.179} C_VEL
LIN {X 0,Y 233.24,Z 617.654,A -85,B 0,C 180,E1 -20441.736,E2 -20441.736} C_VEL
LIN {X 0,Y 229.783,Z 628.399,A -85,B 0,C 180,E1 -20444.616,E2 -20444.616} C_VEL
LIN {X 0,Y 227.055,Z 636.754,A -85,B 0,C 180,E1 -20447.363,E2 -20447.363} C_VEL
LIN {X 0,Y 224.361,Z 644.943,A -85,B 0,C 180,E1 -20450.634,E2 -20450.634} C_VEL
LIN {X 0,Y 222.512,Z 651.068,A -85,B 0,C 180,E1 -20453.655,E2 -20453.655} C_VEL
LIN {X 0,Y 220.888,Z 656.583,A -85,B 0,C 180,E1 -20457.014,E2 -20457.014} C_VEL
LIN {X 0,Y 219.673,Z 661.314,A -85,B 0,C 180,E1 -20460.79,E2 -20460.79} C_VEL
LIN {X 0,Y 219.018,Z 663.809,A -85,B 0,C 180,E1 -20463.455,E2 -20463.455} C_VEL
LIN {X 0,Y 218.518,Z 666.495,A -85,B 0,C 180,E1 -20467.668,E2 -20467.668} C_VEL
LIN {X 0,Y 218.476,Z 667.357,A -85,B 0,C 180,E1 -20470.044,E2 -20470.044} C_VEL
LIN {X 0,Y 218.628,Z 667.764,A -85,B 0,C 180,E1 -20472.459,E2 -20472.459} C_VEL
LIN {X 0,Y 218.942,Z 667.624,A -85,B 0,C 180,E1 -20475.072,E2 -20475.072} C_VEL
LIN {X 0,Y 219.508,Z 666.905,A -85,B 0,C 180,E1 -20477.75,E2 -20477.75} C_VEL
LIN {X 0,Y 220.318,Z 665.659,A -85,B 0,C 180,E1 -20480.357,E2 -20480.357} C_VEL
LIN {X 0,Y 222.028,Z 662.787,A -85,B 0,C 180,E1 -20484.12,E2 -20484.12} C_VEL
LIN {X 0,Y 224.388,Z 658.654,A -85,B 0,C 180,E1 -20487.828,E2 -20487.828} C_VEL
LIN {X 0,Y 227.498,Z 653.171,A -85,B 0,C 180,E1 -20491.444,E2 -20491.444} C_VEL
LIN {X 0,Y 231.127,Z 646.547,A -85,B 0,C 180,E1 -20494.804,E2 -20494.804} C_VEL
LIN {X 0,Y 235.207,Z 638.938,A -85,B 0,C 180,E1 -20497.862,E2 -20497.862} C_VEL
LIN {X 0,Y 239.795,Z 629.927,A -85,B 0,C 180,E1 -20500.754,E2 -20500.754} C_VEL
LIN {X 0,Y 244.358,Z 620.21,A -85,B 0,C 180,E1 -20503.284,E2 -20503.284} C_VEL
LIN {X 0,Y 249.436,Z 608.511,A -85,B 0,C 180,E1 -20505.727,E2 -20505.727} C_VEL
LIN {X 0,Y 254.169,Z 596.246,A -85,B 0,C 180,E1 -20507.801,E2 -20507.801} C_VEL
LIN {X 0,Y 255.601,Z 592.267,A -85,B 0,C 180,E1 -20508.387,E2 -20508.387} C_VEL
LIN {X 0,Y 255.309,Z 587.749,A -85,B 0,C 180,E1 -20509.483,E2 -20509.483} C_VEL
LIN {X 0,Y 253.727,Z 578.034,A -85,B 0,C 180,E1 -20512.039,E2 -20512.039} C_VEL
LIN {X 0,Y 251.382,Z 569.963,A -85,B 0,C 180,E1 -20514.41,E2 -20514.41} C_VEL
LIN {X 0,Y 249.204,Z 563.992,A -85,B 0,C 180,E1 -20516.361,E2 -20516.361} C_VEL
LIN {X 0,Y 244.627,Z 555.057,A -85,B 0,C 180,E1 -20519.999,E2 -20519.999} C_VEL
LIN {X 0,Y 242.702,Z 551.496,A -85,B 0,C 180,E1 -20521.659,E2 -20521.659} C_VEL
LIN {X 0,Y 239.627,Z 547.184,A -85,B 0,C 180,E1 -20524.304,E2 -20524.304} C_VEL
LIN {X 0,Y 237.398,Z 544.659,A -85,B 0,C 180,E1 -20526.348,E2 -20526.348} C_VEL
LIN {X 0,Y 236.521,Z 542.849,A -85,B 0,C 180,E1 -20527.469,E2 -20527.469} C_VEL
LIN {X 0,Y 233.99,Z 540.677,A -85,B 0,C 180,E1 -20530.489,E2 -20530.489} C_VEL
LIN {X 0,Y 232.83,Z 538.475,A -85,B 0,C 180,E1 -20532.64,E2 -20532.64} C_VEL
LIN {X 0,Y 230.808,Z 538.391,A -85,B 0,C 180,E1 -20537.727,E2 -20537.727} C_VEL
LIN {X 0,Y 230.789,Z 539.504,A -85,B 0,C 180,E1 -20542.071,E2 -20542.071} C_VEL
LIN {X 0,Y 233.045,Z 542.526,A -85,B 0,C 180,E1 -20547.502,E2 -20547.502} C_VEL
LIN {X 0,Y 234.884,Z 547.42,A -85,B 0,C 180,E1 -20550.574,E2 -20550.574} C_VEL
LIN {X 0,Y 237.133,Z 550.518,A -85,B 0,C 180,E1 -20552.996,E2 -20552.996} C_VEL
LIN {X 0,Y 238.94,Z 554.859,A -85,B 0,C 180,E1 -20554.978,E2 -20554.978} C_VEL
LIN {X 0,Y 240.011,Z 556.323,A -85,B 0,C 180,E1 -20555.848,E2 -20555.848} C_VEL
LIN {X 0,Y 243.259,Z 563.429,A -85,B 0,C 180,E1 -20558.734,E2 -20558.734} C_VEL
LIN {X 0,Y 245.567,Z 569.273,A -85,B 0,C 180,E1 -20560.715,E2 -20560.715} C_VEL
LIN {X 0,Y 247.562,Z 574.912,A -85,B 0,C 180,E1 -20562.429,E2 -20562.429} C_VEL
LIN {X 0,Y 248.681,Z 580.51,A -85,B 0,C 180,E1 -20563.784,E2 -20563.784} C_VEL
LIN {X 0,Y 248.978,Z 584.944,A -85,B 0,C 180,E1 -20564.674,E2 -20564.674} C_VEL
LIN {X 0,Y 248.408,Z 589.87,A -85,B 0,C 180,E1 -20565.429,E2 -20565.429} C_VEL
LIN {X 0,Y 245.394,Z 603.438,A -85,B 0,C 180,E1 -20567.34,E2 -20567.34} C_VEL
LIN {X 0,Y 245.004,Z 606.477,A -85,B 0,C 180,E1 -20567.928,E2 -20567.928} C_VEL
LIN {X 0,Y 244.001,Z 617.267,A -85,B 0,C 180,E1 -20570.224,E2 -20570.224} C_VEL
LIN {X 0,Y 242.643,Z 624.647,A -85,B 0,C 180,E1 -20571.797,E2 -20571.797} C_VEL
LIN {X 0,Y 237.893,Z 635.364,A -85,B 0,C 180,E1 -20573.782,E2 -20573.782} C_VEL
LIN {X 0,Y 232.385,Z 647.053,A -85,B 0,C 180,E1 -20576.5,E2 -20576.5} C_VEL
LIN {X 0,Y 227.458,Z 656.935,A -85,B 0,C 180,E1 -20579.348,E2 -20579.348} C_VEL
LIN {X 0,Y 223.271,Z 665.241,A -85,B 0,C 180,E1 -20582.335,E2 -20582.335} C_VEL
LIN {X 0,Y 219.657,Z 672.233,A -85,B 0,C 180,E1 -20585.421,E2 -20585.421} C_VEL
LIN {X 0,Y 216.476,Z 678.854,A -85,B 0,C 180,E1 -20589.076,E2 -20589.076} C_VEL
LIN {X 0,Y 214.036,Z 684.13,A -85,B 0,C 180,E1 -20592.811,E2 -20592.811} C_VEL
LIN {X 0,Y 212.488,Z 688.164,A -85,B 0,C 180,E1 -20596.612,E2 -20596.612} C_VEL
LIN {X 0,Y 211.738,Z 691,A -85,B 0,C 180,E1 -20600.446,E2 -20600.446} C_VEL
LIN {X 0,Y 211.696,Z 692.83,A -85,B 0,C 180,E1 -20604.839,E2 -20604.839} C_VEL
LIN {X 0,Y 211.789,Z 693.153,A -85,B 0,C 180,E1 -20608.097,E2 -20608.097} C_VEL
LIN {X 0,Y 211.877,Z 692.964,A -85,B 0,C 180,E1 -20609.999,E2 -20609.999} C_VEL
LIN {X 0,Y 211.766,Z 691.658,A -85,B 0,C 180,E1 -20613.805,E2 -20613.805} C_VEL
LIN {X 0,Y 211.801,Z 690.545,A -85,B 0,C 180,E1 -20615.712,E2 -20615.712} C_VEL
LIN {X 0,Y 211.821,Z 687.305,A -85,B 0,C 180,E1 -20619.548,E2 -20619.548} C_VEL
LIN {X 0,Y 212.507,Z 682.723,A -85,B 0,C 180,E1 -20623.384,E2 -20623.384} C_VEL
LIN {X 0,Y 213.896,Z 676.699,A -85,B 0,C 180,E1 -20627.199,E2 -20627.199} C_VEL
LIN {X 0,Y 216.093,Z 669.088,A -85,B 0,C 180,E1 -20630.961,E2 -20630.961} C_VEL
LIN {X 0,Y 218.813,Z 660.933,A -85,B 0,C 180,E1 -20634.173,E2 -20634.173} C_VEL
LIN {X 0,Y 221.578,Z 652.365,A -85,B 0,C 180,E1 -20636.954,E2 -20636.954} C_VEL
LIN {X 0,Y 224.65,Z 642.87,A -85,B 0,C 180,E1 -20639.518,E2 -20639.518} C_VEL
LIN {X 0,Y 228.371,Z 631.345,A -85,B 0,C 180,E1 -20642.062,E2 -20642.062} C_VEL
LIN {X 0,Y 231.438,Z 621.218,A -85,B 0,C 180,E1 -20643.915,E2 -20643.915} C_VEL
LIN {X 0,Y 232.483,Z 617.409,A -85,B 0,C 180,E1 -20644.527,E2 -20644.527} C_VEL
LIN {X 0,Y 232.164,Z 605.26,A -85,B 0,C 180,E1 -20646.715,E2 -20646.715} C_VEL
LIN {X 0,Y 231.078,Z 592.562,A -85,B 0,C 180,E1 -20648.8,E2 -20648.8} C_VEL
LIN {X 0,Y 229.198,Z 579.244,A -85,B 0,C 180,E1 -20650.797,E2 -20650.797} C_VEL
LIN {X 0,Y 226.212,Z 564.963,A -85,B 0,C 180,E1 -20652.78,E2 -20652.78} C_VEL
LIN {X 0,Y 222.464,Z 551.879,A -85,B 0,C 180,E1 -20654.539,E2 -20654.539} C_VEL
LIN {X 0,Y 219.745,Z 544.798,A -85,B 0,C 180,E1 -20655.545,E2 -20655.545} C_VEL
LIN {X 0,Y 218.067,Z 541.095,A -85,B 0,C 180,E1 -20656.104,E2 -20656.104} C_VEL
LIN {X 0,Y 216.629,Z 538.097,A -85,B 0,C 180,E1 -20656.565,E2 -20656.565} C_VEL
LIN {X 0,Y 216.364,Z 536.837,A -85,B 0,C 180,E1 -20656.745,E2 -20656.745} C_VEL
LIN {X 0,Y 215.449,Z 532.608,A -85,B 0,C 180,E1 -20661.523,E2 -20661.523} C_VEL
LIN {X 0,Y 214.804,Z 528.85,A -85,B 0,C 180,E1 -20666.207,E2 -20666.207} C_VEL
LIN {X 0,Y 214.312,Z 525.475,A -85,B 0,C 180,E1 -20670.535,E2 -20670.535} C_VEL
LIN {X 0,Y 213.831,Z 522.476,A -85,B 0,C 180,E1 -20674.836,E2 -20674.836} C_VEL
LIN {X 0,Y 213.796,Z 522.481,A -85,B 0,C 180,E1 -20678.802,E2 -20678.802} C_VEL
LIN {X 0,Y 213.937,Z 522.461,A -85,B 0,C 180,E1 -20682.804,E2 -20682.804} C_VEL
LIN {X 0,Y 213.974,Z 522.456,A -85,B 0,C 180,E1 -20686.709,E2 -20686.709} C_VEL
LIN {X 0,Y 214.16,Z 522.408,A -85,B 0,C 180,E1 -20690.557,E2 -20690.557} C_VEL
LIN {X 0,Y 214.233,Z 522.409,A -85,B 0,C 180,E1 -20692.461,E2 -20692.461} C_VEL
LIN {X 0,Y 214.442,Z 522.389,A -85,B 0,C 180,E1 -20698.123,E2 -20698.123} C_VEL
LIN {X 0,Y 214.544,Z 522.359,A -85,B 0,C 180,E1 -20700.001,E2 -20700.001} C_VEL
LIN {X 0,Y 214.44,Z 522.371,A -85,B 0,C 180,E1 -20701.879,E2 -20701.879} C_VEL
LIN {X 0,Y 214.203,Z 522.426,A -85,B 0,C 180,E1 -20707.542,E2 -20707.542} C_VEL
LIN {X 0,Y 213.993,Z 522.423,A -85,B 0,C 180,E1 -20711.366,E2 -20711.366} C_VEL
LIN {X 0,Y 213.926,Z 522.45,A -85,B 0,C 180,E1 -20715.238,E2 -20715.238} C_VEL
LIN {X 0,Y 213.863,Z 522.47,A -85,B 0,C 180,E1 -20719.186,E2 -20719.186} C_VEL
LIN {X 0,Y 213.843,Z 522.441,A -85,B 0,C 180,E1 -20723.228,E2 -20723.228} C_VEL
LIN {X 0,Y 213.825,Z 522.465,A -85,B 0,C 180,E1 -20727.451,E2 -20727.451} C_VEL
LIN {X 0,Y 213.776,Z 522.475,A -85,B 0,C 180,E1 -20731.737,E2 -20731.737} C_VEL
LIN {X 0,Y 213.751,Z 522.455,A -85,B 0,C 180,E1 -20736.288,E2 -20736.288} C_VEL
LIN {X 0,Y 213.822,Z 522.476,A -85,B 0,C 180,E1 -20741.101,E2 -20741.101} C_VEL
LIN {X 0,Y 213.835,Z 522.464,A -85,B 0,C 180,E1 -20743.695,E2 -20743.695} C_VEL
LIN {X 0,Y 213.839,Z 522.448,A -85,B 0,C 180,E1 -20746.358,E2 -20746.358} C_VEL
LIN {X 0,Y 213.783,Z 522.485,A -85,B 0,C 180,E1 -20751.348,E2 -20751.348} C_VEL
LIN {X 0,Y 213.769,Z 522.465,A -85,B 0,C 180,E1 -20756.022,E2 -20756.022} C_VEL
LIN {X 0,Y 213.782,Z 522.483,A -85,B 0,C 180,E1 -20760.456,E2 -20760.456} C_VEL
LIN {X 0,Y 213.804,Z 522.468,A -85,B 0,C 180,E1 -20764.704,E2 -20764.704} C_VEL
LIN {X 0,Y 213.816,Z 522.47,A -85,B 0,C 180,E1 -20768.805,E2 -20768.805} C_VEL
LIN {X 0,Y 213.947,Z 522.46,A -85,B 0,C 180,E1 -20772.805,E2 -20772.805} C_VEL
LIN {X 0,Y 213.983,Z 522.449,A -85,B 0,C 180,E1 -20776.71,E2 -20776.71} C_VEL
LIN {X 0,Y 214.143,Z 522.426,A -85,B 0,C 180,E1 -20780.556,E2 -20780.556} C_VEL
LIN {X 0,Y 214.161,Z 522.468,A -85,B 0,C 180,E1 -20783.347,E2 -20783.347} C_VEL
LIN {X 0,Y 215.203,Z 525.387,A -85,B 0,C 180,E1 -20783.755,E2 -20783.755} C_VEL
LIN {X 0,Y 216.601,Z 527.494,A -85,B 0,C 180,E1 -20784.211,E2 -20784.211} C_VEL
LIN {X 0,Y 224.089,Z 540.316,A -85,B 0,C 180,E1 -20786.78,E2 -20786.78} C_VEL
LIN {X 0,Y 227.859,Z 548.921,A -85,B 0,C 180,E1 -20788.359,E2 -20788.359} C_VEL
LIN {X 0,Y 232.593,Z 560.793,A -85,B 0,C 180,E1 -20790.57,E2 -20790.57} C_VEL
LIN {X 0,Y 235.52,Z 573.091,A -85,B 0,C 180,E1 -20792.779,E2 -20792.779} C_VEL
LIN {X 0,Y 237.079,Z 580.874,A -85,B 0,C 180,E1 -20794.251,E2 -20794.251} C_VEL
LIN {X 0,Y 234.328,Z 592.432,A -85,B 0,C 180,E1 -20795.967,E2 -20795.967} C_VEL
LIN {X 0,Y 230.948,Z 604.446,A -85,B 0,C 180,E1 -20798.092,E2 -20798.092} C_VEL
LIN {X 0,Y 227.171,Z 616.503,A -85,B 0,C 180,E1 -20800.698,E2 -20800.698} C_VEL
LIN {X 0,Y 223.672,Z 627.032,A -85,B 0,C 180,E1 -20803.502,E2 -20803.502} C_VEL
LIN {X 0,Y 220.411,Z 636.7,A -85,B 0,C 180,E1 -20806.677,E2 -20806.677} C_VEL
LIN {X 0,Y 217.987,Z 643.86,A -85,B 0,C 180,E1 -20809.545,E2 -20809.545} C_VEL
LIN {X 0,Y 215.741,Z 650.927,A -85,B 0,C 180,E1 -20813.012,E2 -20813.012} C_VEL
LIN {X 0,Y 214.059,Z 656.311,A -85,B 0,C 180,E1 -20816.286,E2 -20816.286} C_VEL
LIN {X 0,Y 212.869,Z 660.646,A -85,B 0,C 180,E1 -20819.686,E2 -20819.686} C_VEL
LIN {X 0,Y 212.241,Z 663.016,A -85,B 0,C 180,E1 -20821.993,E2 -20821.993} C_VEL
LIN {X 0,Y 211.736,Z 664.969,A -85,B 0,C 180,E1 -20824.352,E2 -20824.352} C_VEL
LIN {X 0,Y 211.451,Z 666.605,A -85,B 0,C 180,E1 -20827.088,E2 -20827.088} C_VEL
LIN {X 0,Y 211.397,Z 667.758,A -85,B 0,C 180,E1 -20830.123,E2 -20830.123} C_VEL
LIN {X 0,Y 211.709,Z 668.184,A -85,B 0,C 180,E1 -20834.197,E2 -20834.197} C_VEL
LIN {X 0,Y 212.173,Z 667.817,A -85,B 0,C 180,E1 -20836.78,E2 -20836.78} C_VEL
LIN {X 0,Y 212.901,Z 666.919,A -85,B 0,C 180,E1 -20839.398,E2 -20839.398} C_VEL
LIN {X 0,Y 213.889,Z 665.413,A -85,B 0,C 180,E1 -20842.055,E2 -20842.055} C_VEL
LIN {X 0,Y 215.241,Z 663.332,A -85,B 0,C 180,E1 -20844.716,E2 -20844.716} C_VEL
LIN {X 0,Y 216.929,Z 660.641,A -85,B 0,C 180,E1 -20847.388,E2 -20847.388} C_VEL
LIN {X 0,Y 220.262,Z 655.206,A -85,B 0,C 180,E1 -20851.404,E2 -20851.404} C_VEL
LIN {X 0,Y 223.664,Z 649.471,A -85,B 0,C 180,E1 -20854.617,E2 -20854.617} C_VEL
LIN {X 0,Y 227.722,Z 642.334,A -85,B 0,C 180,E1 -20857.799,E2 -20857.799} C_VEL
LIN {X 0,Y 231.976,Z 634.664,A -85,B 0,C 180,E1 -20860.533,E2 -20860.533} C_VEL
LIN {X 0,Y 237.093,Z 624.695,A -85,B 0,C 180,E1 -20863.422,E2 -20863.422} C_VEL
LIN {X 0,Y 241.957,Z 614.431,A -85,B 0,C 180,E1 -20865.815,E2 -20865.815} C_VEL
LIN {X 0,Y 246.689,Z 603.403,A -85,B 0,C 180,E1 -20867.911,E2 -20867.911} C_VEL
LIN {X 0,Y 250.19,Z 594.369,A -85,B 0,C 180,E1 -20869.335,E2 -20869.335} C_VEL
LIN {X 0,Y 249.259,Z 585.015,A -85,B 0,C 180,E1 -20871.895,E2 -20871.895} C_VEL
LIN {X 0,Y 247.654,Z 577.546,A -85,B 0,C 180,E1 -20874.122,E2 -20874.122} C_VEL
LIN {X 0,Y 245.259,Z 569.789,A -85,B 0,C 180,E1 -20876.714,E2 -20876.714} C_VEL
LIN {X 0,Y 241.648,Z 562.02,A -85,B 0,C 180,E1 -20879.999,E2 -20879.999} C_VEL
LIN {X 0,Y 239.966,Z 558.398,A -85,B 0,C 180,E1 -20881.678,E2 -20881.678} C_VEL
LIN {X 0,Y 237.208,Z 554,A -85,B 0,C 180,E1 -20884.348,E2 -20884.348} C_VEL
LIN {X 0,Y 235.419,Z 552.085,A -85,B 0,C 180,E1 -20886.037,E2 -20886.037} C_VEL
LIN {X 0,Y 234.108,Z 549.466,A -85,B 0,C 180,E1 -20887.833,E2 -20887.833} C_VEL
LIN {X 0,Y 231.193,Z 546.244,A -85,B 0,C 180,E1 -20892.058,E2 -20892.058} C_VEL
LIN {X 0,Y 230.825,Z 545.26,A -85,B 0,C 180,E1 -20893.016,E2 -20893.016} C_VEL
LIN {X 0,Y 228.954,Z 545.436,A -85,B 0,C 180,E1 -20898.802,E2 -20898.802} C_VEL
LIN {X 0,Y 229.306,Z 546.925,A -85,B 0,C 180,E1 -20903.151,E2 -20903.151} C_VEL
LIN {X 0,Y 231.052,Z 549.34,A -85,B 0,C 180,E1 -20907.222,E2 -20907.222} C_VEL
LIN {X 0,Y 232.317,Z 553.442,A -85,B 0,C 180,E1 -20909.838,E2 -20909.838} C_VEL
LIN {X 0,Y 234.569,Z 557.174,A -85,B 0,C 180,E1 -20912.636,E2 -20912.636} C_VEL
LIN {X 0,Y 236.03,Z 560.958,A -85,B 0,C 180,E1 -20914.453,E2 -20914.453} C_VEL
LIN {X 0,Y 236.976,Z 562.38,A -85,B 0,C 180,E1 -20915.331,E2 -20915.331} C_VEL
LIN {X 0,Y 239.609,Z 568.753,A -85,B 0,C 180,E1 -20918.02,E2 -20918.02} C_VEL
LIN {X 0,Y 242.348,Z 576.441,A -85,B 0,C 180,E1 -20920.73,E2 -20920.73} C_VEL
LIN {X 0,Y 243.22,Z 579.426,A -85,B 0,C 180,E1 -20921.651,E2 -20921.651} C_VEL
LIN {X 0,Y 244.41,Z 587.353,A -85,B 0,C 180,E1 -20923.639,E2 -20923.639} C_VEL
LIN {X 0,Y 245.157,Z 598.95,A -85,B 0,C 180,E1 -20926.308,E2 -20926.308} C_VEL
LIN {X 0,Y 245.004,Z 606.477,A -85,B 0,C 180,E1 -20927.928,E2 -20927.928} C_VEL
LIN {X 0,Y 244.135,Z 611.141,A -85,B 0,C 180,E1 -20928.775,E2 -20928.775} C_VEL
LIN {X 0,Y 242.399,Z 615.922,A -85,B 0,C 180,E1 -20929.492,E2 -20929.492} C_VEL
LIN {X 0,Y 237.512,Z 625.472,A -85,B 0,C 180,E1 -20930.829,E2 -20930.829} C_VEL
LIN {X 0,Y 234.371,Z 631.559,A -85,B 0,C 180,E1 -20931.866,E2 -20931.866} C_VEL
LIN {X 0,Y 229.772,Z 641.195,A -85,B 0,C 180,E1 -20933.928,E2 -20933.928} C_VEL
LIN {X 0,Y 224.247,Z 651.873,A -85,B 0,C 180,E1 -20936.738,E2 -20936.738} C_VEL
LIN {X 0,Y 219.329,Z 660.966,A -85,B 0,C 180,E1 -20939.729,E2 -20939.729} C_VEL
LIN {X 0,Y 215.335,Z 668.479,A -85,B 0,C 180,E1 -20942.811,E2 -20942.811} C_VEL
LIN {X 0,Y 211.345,Z 675.706,A -85,B 0,C 180,E1 -20946.481,E2 -20946.481} C_VEL
LIN {X 0,Y 208.346,Z 681.518,A -85,B 0,C 180,E1 -20950.285,E2 -20950.285} C_VEL
LIN {X 0,Y 206.24,Z 686.072,A -85,B 0,C 180,E1 -20954.179,E2 -20954.179} C_VEL
LIN {X 0,Y 204.997,Z 689.435,A -85,B 0,C 180,E1 -20958.129,E2 -20958.129} C_VEL
LIN {X 0,Y 204.525,Z 691.622,A -85,B 0,C 180,E1 -20962.099,E2 -20962.099} C_VEL
LIN {X 0,Y 204.59,Z 692.63,A -85,B 0,C 180,E1 -20966.06,E2 -20966.06} C_VEL
LIN {X 0,Y 204.717,Z 692.704,A -85,B 0,C 180,E1 -20968.032,E2 -20968.032} C_VEL
LIN {X 0,Y 204.805,Z 692.479,A -85,B 0,C 180,E1 -20969.999,E2 -20969.999} C_VEL
LIN {X 0,Y 204.691,Z 691.101,A -85,B 0,C 180,E1 -20973.936,E2 -20973.936} C_VEL
LIN {X 0,Y 204.7,Z 689.948,A -85,B 0,C 180,E1 -20975.911,E2 -20975.911} C_VEL
LIN {X 0,Y 204.773,Z 686.66,A -85,B 0,C 180,E1 -20979.88,E2 -20979.88} C_VEL
LIN {X 0,Y 205.541,Z 682.009,A -85,B 0,C 180,E1 -20983.847,E2 -20983.847} C_VEL
LIN {X 0,Y 207.031,Z 675.897,A -85,B 0,C 180,E1 -20987.788,E2 -20987.788} C_VEL
LIN {X 0,Y 209.364,Z 668.188,A -85,B 0,C 180,E1 -20991.668,E2 -20991.668} C_VEL
LIN {X 0,Y 212.251,Z 659.933,A -85,B 0,C 180,E1 -20994.97,E2 -20994.97} C_VEL
LIN {X 0,Y 214.981,Z 651.669,A -85,B 0,C 180,E1 -20997.7,E2 -20997.7} C_VEL
LIN {X 0,Y 218.394,Z 641.614,A -85,B 0,C 180,E1 -21000.452,E2 -21000.452} C_VEL
LIN {X 0,Y 222.235,Z 629.918,A -85,B 0,C 180,E1 -21003.058,E2 -21003.058} C_VEL
LIN {X 0,Y 225.747,Z 618.812,A -85,B 0,C 180,E1 -21005.072,E2 -21005.072} C_VEL
LIN {X 0,Y 225.764,Z 608.243,A -85,B 0,C 180,E1 -21007.071,E2 -21007.071} C_VEL
LIN {X 0,Y 224.81,Z 594.857,A -85,B 0,C 180,E1 -21009.4,E2 -21009.4} C_VEL
LIN {X 0,Y 223.2,Z 582.245,A -85,B 0,C 180,E1 -21011.392,E2 -21011.392} C_VEL
LIN {X 0,Y 220.459,Z 567.936,A -85,B 0,C 180,E1 -21013.512,E2 -21013.512} C_VEL
LIN {X 0,Y 216.578,Z 553.758,A -85,B 0,C 180,E1 -21015.559,E2 -21015.559} C_VEL
LIN {X 0,Y 213.341,Z 545.736,A -85,B 0,C 180,E1 -21016.798,E2 -21016.798} C_VEL
LIN {X 0,Y 211.441,Z 541.615,A -85,B 0,C 180,E1 -21017.454,E2 -21017.454} C_VEL
LIN {X 0,Y 209.479,Z 538.099,A -85,B 0,C 180,E1 -21018.099,E2 -21018.099} C_VEL
LIN {X 0,Y 209.056,Z 536.354,A -85,B 0,C 180,E1 -21018.318,E2 -21018.318} C_VEL
LIN {X 0,Y 208.053,Z 531.61,A -85,B 0,C 180,E1 -21024.163,E2 -21024.163} C_VEL
LIN {X 0,Y 207.42,Z 527.51,A -85,B 0,C 180,E1 -21029.454,E2 -21029.454} C_VEL
LIN {X 0,Y 206.967,Z 524.477,A -85,B 0,C 180,E1 -21033.805,E2 -21033.805} C_VEL
LIN {X 0,Y 206.781,Z 523.353,A -85,B 0,C 180,E1 -21035.664,E2 -21035.664} C_VEL
LIN {X 0,Y 206.771,Z 523.356,A -85,B 0,C 180,E1 -21040.13,E2 -21040.13} C_VEL
LIN {X 0,Y 206.86,Z 523.343,A -85,B 0,C 180,E1 -21044.229,E2 -21044.229} C_VEL
LIN {X 0,Y 207.09,Z 523.291,A -85,B 0,C 180,E1 -21049.781,E2 -21049.781} C_VEL
LIN {X 0,Y 207.171,Z 523.284,A -85,B 0,C 180,E1 -21052.202,E2 -21052.202} C_VEL
LIN {X 0,Y 207.378,Z 523.268,A -85,B 0,C 180,E1 -21058.059,E2 -21058.059} C_VEL
LIN {X 0,Y 207.509,Z 523.233,A -85,B 0,C 180,E1 -21060.001,E2 -21060.001} C_VEL
LIN {X 0,Y 207.377,Z 523.25,A -85,B 0,C 180,E1 -21061.943,E2 -21061.943} C_VEL
LIN {X 0,Y 207.143,Z 523.304,A -85,B 0,C 180,E1 -21067.801,E2 -21067.801} C_VEL
LIN {X 0,Y 206.917,Z 523.3,A -85,B 0,C 180,E1 -21071.76,E2 -21071.76} C_VEL
LIN {X 0,Y 206.86,Z 523.333,A -85,B 0,C 180,E1 -21075.772,E2 -21075.772} C_VEL
LIN {X 0,Y 206.794,Z 523.345,A -85,B 0,C 180,E1 -21079.869,E2 -21079.869} C_VEL
LIN {X 0,Y 206.759,Z 523.319,A -85,B 0,C 180,E1 -21084.074,E2 -21084.074} C_VEL
LIN {X 0,Y 206.74,Z 523.354,A -85,B 0,C 180,E1 -21088.42,E2 -21088.42} C_VEL
LIN {X 0,Y 206.706,Z 523.348,A -85,B 0,C 180,E1 -21092.957,E2 -21092.957} C_VEL
LIN {X 0,Y 206.723,Z 523.341,A -85,B 0,C 180,E1 -21097.732,E2 -21097.732} C_VEL
LIN {X 0,Y 206.748,Z 523.358,A -85,B 0,C 180,E1 -21101.598,E2 -21101.598} C_VEL
LIN {X 0,Y 206.744,Z 523.331,A -85,B 0,C 180,E1 -21105.552,E2 -21105.552} C_VEL
LIN {X 0,Y 206.727,Z 523.359,A -85,B 0,C 180,E1 -21109.767,E2 -21109.767} C_VEL
LIN {X 0,Y 206.726,Z 523.36,A -85,B 0,C 180,E1 -21112.272,E2 -21112.272} C_VEL
LIN {X 0,Y 206.71,Z 523.351,A -85,B 0,C 180,E1 -21117.046,E2 -21117.046} C_VEL
LIN {X 0,Y 206.768,Z 523.348,A -85,B 0,C 180,E1 -21122.098,E2 -21122.098} C_VEL
LIN {X 0,Y 206.788,Z 523.353,A -85,B 0,C 180,E1 -21126.585,E2 -21126.585} C_VEL
LIN {X 0,Y 206.877,Z 523.339,A -85,B 0,C 180,E1 -21132.198,E2 -21132.198} C_VEL
LIN {X 0,Y 206.917,Z 523.326,A -85,B 0,C 180,E1 -21136.247,E2 -21136.247} C_VEL
LIN {X 0,Y 207.119,Z 523.303,A -85,B 0,C 180,E1 -21141.218,E2 -21141.218} C_VEL
LIN {X 0,Y 207.126,Z 523.307,A -85,B 0,C 180,E1 -21141.771,E2 -21141.771} C_VEL
LIN {X 0,Y 208.092,Z 526.075,A -85,B 0,C 180,E1 -21142.207,E2 -21142.207} C_VEL
LIN {X 0,Y 209.664,Z 528.324,A -85,B 0,C 180,E1 -21142.751,E2 -21142.751} C_VEL
LIN {X 0,Y 215.91,Z 539.175,A -85,B 0,C 180,E1 -21145.038,E2 -21145.038} C_VEL
LIN {X 0,Y 219.94,Z 546.708,A -85,B 0,C 180,E1 -21146.615,E2 -21146.615} C_VEL
LIN {X 0,Y 225.731,Z 561.295,A -85,B 0,C 180,E1 -21149.465,E2 -21149.465} C_VEL
LIN {X 0,Y 227.799,Z 568.438,A -85,B 0,C 180,E1 -21150.823,E2 -21150.823} C_VEL
LIN {X 0,Y 230.275,Z 580.423,A -85,B 0,C 180,E1 -21153.144,E2 -21153.144} C_VEL
LIN {X 0,Y 230.583,Z 583.401,A -85,B 0,C 180,E1 -21153.714,E2 -21153.714} C_VEL
LIN {X 0,Y 227.225,Z 595.792,A -85,B 0,C 180,E1 -21155.625,E2 -21155.625} C_VEL
LIN {X 0,Y 223.669,Z 607.788,A -85,B 0,C 180,E1 -21157.902,E2 -21157.902} C_VEL
LIN {X 0,Y 220.221,Z 618.3,A -85,B 0,C 180,E1 -21160.323,E2 -21160.323} C_VEL
LIN {X 0,Y 216.616,Z 628.755,A -85,B 0,C 180,E1 -21163.257,E2 -21163.257} C_VEL
LIN {X 0,Y 213.372,Z 638.003,A -85,B 0,C 180,E1 -21166.457,E2 -21166.457} C_VEL
LIN {X 0,Y 210.441,Z 646.248,A -85,B 0,C 180,E1 -21169.985,E2 -21169.985} C_VEL
LIN {X 0,Y 208.702,Z 651.574,A -85,B 0,C 180,E1 -21172.785,E2 -21172.785} C_VEL
LIN {X 0,Y 206.971,Z 656.957,A -85,B 0,C 180,E1 -21176.196,E2 -21176.196} C_VEL
LIN {X 0,Y 205.762,Z 661.232,A -85,B 0,C 180,E1 -21179.688,E2 -21179.688} C_VEL
LIN {X 0,Y 204.624,Z 665.475,A -85,B 0,C 180,E1 -21184.481,E2 -21184.481} C_VEL
LIN {X 0,Y 204.312,Z 667.509,A -85,B 0,C 180,E1 -21188.256,E2 -21188.256} C_VEL
LIN {X 0,Y 204.325,Z 668.335,A -85,B 0,C 180,E1 -21190.823,E2 -21190.823} C_VEL
LIN {X 0,Y 204.576,Z 668.655,A -85,B 0,C 180,E1 -21193.826,E2 -21193.826} C_VEL
LIN {X 0,Y 205.066,Z 668.368,A -85,B 0,C 180,E1 -21196.729,E2 -21196.729} C_VEL
LIN {X 0,Y 205.852,Z 667.536,A -85,B 0,C 180,E1 -21199.557,E2 -21199.557} C_VEL
LIN {X 0,Y 207.863,Z 664.815,A -85,B 0,C 180,E1 -21204.239,E2 -21204.239} C_VEL
LIN {X 0,Y 210.785,Z 660.466,A -85,B 0,C 180,E1 -21208.764,E2 -21208.764} C_VEL
LIN {X 0,Y 214.261,Z 655.174,A -85,B 0,C 180,E1 -21212.662,E2 -21212.662} C_VEL
LIN {X 0,Y 218.358,Z 648.679,A -85,B 0,C 180,E1 -21216.28,E2 -21216.28} C_VEL
LIN {X 0,Y 223.191,Z 640.679,A -85,B 0,C 180,E1 -21219.733,E2 -21219.733} C_VEL
LIN {X 0,Y 228.55,Z 631.29,A -85,B 0,C 180,E1 -21222.902,E2 -21222.902} C_VEL
LIN {X 0,Y 233.129,Z 622.587,A -85,B 0,C 180,E1 -21225.286,E2 -21225.286} C_VEL
LIN {X 0,Y 238.799,Z 610.87,A -85,B 0,C 180,E1 -21227.861,E2 -21227.861} C_VEL
LIN {X 0,Y 244.134,Z 598.429,A -85,B 0,C 180,E1 -21230.053,E2 -21230.053} C_VEL
LIN {X 0,Y 244.688,Z 596.558,A -85,B 0,C 180,E1 -21230.389,E2 -21230.389} C_VEL
LIN {X 0,Y 243.974,Z 587.684,A -85,B 0,C 180,E1 -21232.967,E2 -21232.967} C_VEL
LIN {X 0,Y 242.485,Z 580.139,A -85,B 0,C 180,E1 -21235.428,E2 -21235.428} C_VEL
LIN {X 0,Y 240.883,Z 574.475,A -85,B 0,C 180,E1 -21237.479,E2 -21237.479} C_VEL
LIN {X 0,Y 237.823,Z 567.263,A -85,B 0,C 180,E1 -21240.714,E2 -21240.714} C_VEL
LIN {X 0,Y 235.357,Z 562.208,A -85,B 0,C 180,E1 -21243.423,E2 -21243.423} C_VEL
LIN {X 0,Y 233.744,Z 559.757,A -85,B 0,C 180,E1 -21245.175,E2 -21245.175} C_VEL
LIN {X 0,Y 231.728,Z 556.475,A -85,B 0,C 180,E1 -21247.805,E2 -21247.805} C_VEL
LIN {X 0,Y 228.923,Z 552.8,A -85,B 0,C 180,E1 -21252.409,E2 -21252.409} C_VEL
LIN {X 0,Y 228.176,Z 552.026,A -85,B 0,C 180,E1 -21254.264,E2 -21254.264} C_VEL
LIN {X 0,Y 227.104,Z 552.125,A -85,B 0,C 180,E1 -21258.026,E2 -21258.026} C_VEL
LIN {X 0,Y 227.095,Z 553.139,A -85,B 0,C 180,E1 -21261.81,E2 -21261.81} C_VEL
LIN {X 0,Y 228.135,Z 555.076,A -85,B 0,C 180,E1 -21265.549,E2 -21265.549} C_VEL
LIN {X 0,Y 228.799,Z 556.293,A -85,B 0,C 180,E1 -21267.027,E2 -21267.027} C_VEL
LIN {X 0,Y 229.693,Z 559.701,A -85,B 0,C 180,E1 -21269.311,E2 -21269.311} C_VEL
LIN {X 0,Y 231.489,Z 562.836,A -85,B 0,C 180,E1 -21271.78,E2 -21271.78} C_VEL
LIN {X 0,Y 232.937,Z 566.969,A -85,B 0,C 180,E1 -21273.928,E2 -21273.928} C_VEL
LIN {X 0,Y 233.797,Z 568.415,A -85,B 0,C 180,E1 -21274.829,E2 -21274.829} C_VEL
LIN {X 0,Y 236.347,Z 575.734,A -85,B 0,C 180,E1 -21277.934,E2 -21277.934} C_VEL
LIN {X 0,Y 238.024,Z 580.901,A -85,B 0,C 180,E1 -21279.853,E2 -21279.853} C_VEL
LIN {X 0,Y 238.978,Z 585.199,A -85,B 0,C 180,E1 -21281.204,E2 -21281.204} C_VEL
LIN {X 0,Y 239.719,Z 592.768,A -85,B 0,C 180,E1 -21283.185,E2 -21283.185} C_VEL
LIN {X 0,Y 239.942,Z 603.532,A -85,B 0,C 180,E1 -21285.774,E2 -21285.774} C_VEL
LIN {X 0,Y 239.18,Z 613.26,A -85,B 0,C 180,E1 -21287.967,E2 -21287.967} C_VEL
LIN {X 0,Y 237.54,Z 623.547,A -85,B 0,C 180,E1 -21290.286,E2 -21290.286} C_VEL
LIN {X 0,Y 236.958,Z 625.895,A -85,B 0,C 180,E1 -21290.819,E2 -21290.819} C_VEL
LIN {X 0,Y 234.371,Z 631.559,A -85,B 0,C 180,E1 -21291.866,E2 -21291.866} C_VEL
LIN {X 0,Y 231.835,Z 635.923,A -85,B 0,C 180,E1 -21292.639,E2 -21292.639} C_VEL
LIN {X 0,Y 226.208,Z 642.813,A -85,B 0,C 180,E1 -21293.734,E2 -21293.734} C_VEL
LIN {X 0,Y 220.51,Z 649.329,A -85,B 0,C 180,E1 -21294.966,E2 -21294.966} C_VEL
LIN {X 0,Y 217.905,Z 653.006,A -85,B 0,C 180,E1 -21295.953,E2 -21295.953} C_VEL
LIN {X 0,Y 213.09,Z 661.407,A -85,B 0,C 180,E1 -21298.84,E2 -21298.84} C_VEL
LIN {X 0,Y 209.002,Z 668.609,A -85,B 0,C 180,E1 -21301.915,E2 -21301.915} C_VEL
LIN {X 0,Y 204.801,Z 675.704,A -85,B 0,C 180,E1 -21305.682,E2 -21305.682} C_VEL
LIN {X 0,Y 201.625,Z 681.416,A -85,B 0,C 180,E1 -21309.6,E2 -21309.6} C_VEL
LIN {X 0,Y 199.343,Z 685.862,A -85,B 0,C 180,E1 -21313.617,E2 -21313.617} C_VEL
LIN {X 0,Y 197.977,Z 689.131,A -85,B 0,C 180,E1 -21317.701,E2 -21317.701} C_VEL
LIN {X 0,Y 197.447,Z 691.27,A -85,B 0,C 180,E1 -21321.814,E2 -21321.814} C_VEL
LIN {X 0,Y 197.499,Z 692.213,A -85,B 0,C 180,E1 -21325.918,E2 -21325.918} C_VEL
LIN {X 0,Y 197.645,Z 692.251,A -85,B 0,C 180,E1 -21327.961,E2 -21327.961} C_VEL
LIN {X 0,Y 197.734,Z 691.991,A -85,B 0,C 180,E1 -21329.999,E2 -21329.999} C_VEL
LIN {X 0,Y 197.619,Z 690.542,A -85,B 0,C 180,E1 -21334.078,E2 -21334.078} C_VEL
LIN {X 0,Y 197.592,Z 689.35,A -85,B 0,C 180,E1 -21336.124,E2 -21336.124} C_VEL
LIN {X 0,Y 197.717,Z 685.987,A -85,B 0,C 180,E1 -21340.236,E2 -21340.236} C_VEL
LIN {X 0,Y 198.589,Z 681.277,A -85,B 0,C 180,E1 -21344.342,E2 -21344.342} C_VEL
LIN {X 0,Y 200.19,Z 675.083,A -85,B 0,C 180,E1 -21348.417,E2 -21348.417} C_VEL
LIN {X 0,Y 202.703,Z 667.261,A -85,B 0,C 180,E1 -21352.418,E2 -21352.418} C_VEL
LIN {X 0,Y 205.717,Z 658.924,A -85,B 0,C 180,E1 -21355.821,E2 -21355.821} C_VEL
LIN {X 0,Y 209.246,Z 648.8,A -85,B 0,C 180,E1 -21359.16,E2 -21359.16} C_VEL
LIN {X 0,Y 212.839,Z 638.567,A -85,B 0,C 180,E1 -21361.891,E2 -21361.891} C_VEL
LIN {X 0,Y 216.563,Z 627.432,A -85,B 0,C 180,E1 -21364.321,E2 -21364.321} C_VEL
LIN {X 0,Y 219.024,Z 620.076,A -85,B 0,C 180,E1 -21365.676,E2 -21365.676} C_VEL
LIN {X 0,Y 219.331,Z 616.644,A -85,B 0,C 180,E1 -21366.34,E2 -21366.34} C_VEL
LIN {X 0,Y 219.06,Z 604.575,A -85,B 0,C 180,E1 -21368.671,E2 -21368.671} C_VEL
LIN {X 0,Y 218.042,Z 591.876,A -85,B 0,C 180,E1 -21370.912,E2 -21370.912} C_VEL
LIN {X 0,Y 215.981,Z 577.578,A -85,B 0,C 180,E1 -21373.242,E2 -21373.242} C_VEL
LIN {X 0,Y 213.411,Z 565.481,A -85,B 0,C 180,E1 -21375.102,E2 -21375.102} C_VEL
LIN {X 0,Y 209.952,Z 553.723,A -85,B 0,C 180,E1 -21376.916,E2 -21376.916} C_VEL
LIN {X 0,Y 205.801,Z 544.741,A -85,B 0,C 180,E1 -21378.518,E2 -21378.518} C_VEL
LIN {X 0,Y 203.759,Z 540.576,A -85,B 0,C 180,E1 -21379.27,E2 -21379.27} C_VEL
LIN {X 0,Y 202.076,Z 537.596,A -85,B 0,C 180,E1 -21379.863,E2 -21379.863} C_VEL
LIN {X 0,Y 201.621,Z 535.886,A -85,B 0,C 180,E1 -21380.114,E2 -21380.114} C_VEL
LIN {X 0,Y 201.102,Z 533.138,A -85,B 0,C 180,E1 -21383.552,E2 -21383.552} C_VEL
LIN {X 0,Y 200.546,Z 529.564,A -85,B 0,C 180,E1 -21388.288,E2 -21388.288} C_VEL
LIN {X 0,Y 200.096,Z 526.431,A -85,B 0,C 180,E1 -21392.833,E2 -21392.833} C_VEL
LIN {X 0,Y 199.725,Z 524.234,A -85,B 0,C 180,E1 -21396.186,E2 -21396.186} C_VEL
LIN {X 0,Y 199.789,Z 524.226,A -85,B 0,C 180,E1 -21401.758,E2 -21401.758} C_VEL
LIN {X 0,Y 199.841,Z 524.218,A -85,B 0,C 180,E1 -21405.749,E2 -21405.749} C_VEL
LIN {X 0,Y 200.064,Z 524.164,A -85,B 0,C 180,E1 -21409.885,E2 -21409.885} C_VEL
LIN {X 0,Y 200.032,Z 524.187,A -85,B 0,C 180,E1 -21413.95,E2 -21413.95} C_VEL
LIN {X 0,Y 200.318,Z 524.148,A -85,B 0,C 180,E1 -21417.99,E2 -21417.99} C_VEL
LIN {X 0,Y 200.473,Z 524.108,A -85,B 0,C 180,E1 -21420.001,E2 -21420.001} C_VEL
LIN {X 0,Y 200.026,Z 524.184,A -85,B 0,C 180,E1 -21424.03,E2 -21424.03} C_VEL
LIN {X 0,Y 200.09,Z 524.181,A -85,B 0,C 180,E1 -21428.077,E2 -21428.077} C_VEL
LIN {X 0,Y 199.868,Z 524.175,A -85,B 0,C 180,E1 -21432.181,E2 -21432.181} C_VEL
LIN {X 0,Y 199.799,Z 524.218,A -85,B 0,C 180,E1 -21436.345,E2 -21436.345} C_VEL
LIN {X 0,Y 199.819,Z 524.218,A -85,B 0,C 180,E1 -21438.455,E2 -21438.455} C_VEL
LIN {X 0,Y 199.732,Z 524.193,A -85,B 0,C 180,E1 -21443.818,E2 -21443.818} C_VEL
LIN {X 0,Y 199.709,Z 524.23,A -85,B 0,C 180,E1 -21448.388,E2 -21448.388} C_VEL
LIN {X 0,Y 199.661,Z 524.231,A -85,B 0,C 180,E1 -21452.354,E2 -21452.354} C_VEL
LIN {X 0,Y 199.651,Z 524.211,A -85,B 0,C 180,E1 -21456.758,E2 -21456.758} C_VEL
LIN {X 0,Y 199.699,Z 524.229,A -85,B 0,C 180,E1 -21459.308,E2 -21459.308} C_VEL
LIN {X 0,Y 199.698,Z 524.232,A -85,B 0,C 180,E1 -21462.352,E2 -21462.352} C_VEL
LIN {X 0,Y 199.692,Z 524.21,A -85,B 0,C 180,E1 -21465.263,E2 -21465.263} C_VEL
LIN {X 0,Y 199.677,Z 524.221,A -85,B 0,C 180,E1 -21468.032,E2 -21468.032} C_VEL
LIN {X 0,Y 199.701,Z 524.237,A -85,B 0,C 180,E1 -21470.738,E2 -21470.738} C_VEL
LIN {X 0,Y 199.634,Z 524.223,A -85,B 0,C 180,E1 -21475.72,E2 -21475.72} C_VEL
LIN {X 0,Y 199.705,Z 524.232,A -85,B 0,C 180,E1 -21478.14,E2 -21478.14} C_VEL
LIN {X 0,Y 199.688,Z 524.223,A -85,B 0,C 180,E1 -21482.774,E2 -21482.774} C_VEL
LIN {X 0,Y 199.741,Z 524.232,A -85,B 0,C 180,E1 -21487.231,E2 -21487.231} C_VEL
LIN {X 0,Y 199.8,Z 524.215,A -85,B 0,C 180,E1 -21491.759,E2 -21491.759} C_VEL
LIN {X 0,Y 199.851,Z 524.204,A -85,B 0,C 180,E1 -21495.751,E2 -21495.751} C_VEL
LIN {X 0,Y 200.085,Z 524.377,A -85,B 0,C 180,E1 -21500.153,E2 -21500.153} C_VEL
LIN {X 0,Y 201.152,Z 527.154,A -85,B 0,C 180,E1 -21500.627,E2 -21500.627} C_VEL
LIN {X 0,Y 202.726,Z 529.317,A -85,B 0,C 180,E1 -21501.194,E2 -21501.194} C_VEL
LIN {X 0,Y 207.516,Z 537.865,A -85,B 0,C 180,E1 -21503.092,E2 -21503.092} C_VEL
LIN {X 0,Y 213.883,Z 549.272,A -85,B 0,C 180,E1 -21505.695,E2 -21505.695} C_VEL
LIN {X 0,Y 217.353,Z 558.015,A -85,B 0,C 180,E1 -21507.482,E2 -21507.482} C_VEL
LIN {X 0,Y 221.093,Z 568.497,A -85,B 0,C 180,E1 -21509.673,E2 -21509.673} C_VEL
LIN {X 0,Y 223.945,Z 582.391,A -85,B 0,C 180,E1 -21512.474,E2 -21512.474} C_VEL
LIN {X 0,Y 224.272,Z 584.473,A -85,B 0,C 180,E1 -21512.92,E2 -21512.92} C_VEL
LIN {X 0,Y 220.558,Z 597.597,A -85,B 0,C 180,E1 -21515.028,E2 -21515.028} C_VEL
LIN {X 0,Y 216.783,Z 609.749,A -85,B 0,C 180,E1 -21517.452,E2 -21517.452} C_VEL
LIN {X 0,Y 212.9,Z 620.991,A -85,B 0,C 180,E1 -21520.196,E2 -21520.196} C_VEL
LIN {X 0,Y 209.33,Z 630.935,A -85,B 0,C 180,E1 -21523.181,E2 -21523.181} C_VEL
LIN {X 0,Y 206.207,Z 639.533,A -85,B 0,C 180,E1 -21526.337,E2 -21526.337} C_VEL
LIN {X 0,Y 203.454,Z 646.984,A -85,B 0,C 180,E1 -21529.683,E2 -21529.683} C_VEL
LIN {X 0,Y 201.141,Z 653.732,A -85,B 0,C 180,E1 -21533.469,E2 -21533.469} C_VEL
LIN {X 0,Y 199.464,Z 659.036,A -85,B 0,C 180,E1 -21537.262,E2 -21537.262} C_VEL
LIN {X 0,Y 198.643,Z 661.794,A -85,B 0,C 180,E1 -21539.691,E2 -21539.691} C_VEL
LIN {X 0,Y 197.972,Z 664.133,A -85,B 0,C 180,E1 -21542.175,E2 -21542.175} C_VEL
LIN {X 0,Y 197.45,Z 666.214,A -85,B 0,C 180,E1 -21545.048,E2 -21545.048} C_VEL
LIN {X 0,Y 197.212,Z 667.917,A -85,B 0,C 180,E1 -21548.37,E2 -21548.37} C_VEL
LIN {X 0,Y 197.351,Z 668.992,A -85,B 0,C 180,E1 -21552.581,E2 -21552.581} C_VEL
LIN {X 0,Y 197.71,Z 669.074,A -85,B 0,C 180,E1 -21555.312,E2 -21555.312} C_VEL
LIN {X 0,Y 198.312,Z 668.662,A -85,B 0,C 180,E1 -21558.092,E2 -21558.092} C_VEL
LIN {X 0,Y 199.219,Z 667.672,A -85,B 0,C 180,E1 -21560.906,E2 -21560.906} C_VEL
LIN {X 0,Y 200.473,Z 666.124,A -85,B 0,C 180,E1 -21563.738,E2 -21563.738} C_VEL
LIN {X 0,Y 202.836,Z 662.973,A -85,B 0,C 180,E1 -21567.707,E2 -21567.707} C_VEL
LIN {X 0,Y 205.863,Z 658.799,A -85,B 0,C 180,E1 -21571.447,E2 -21571.447} C_VEL
LIN {X 0,Y 210.376,Z 652.276,A -85,B 0,C 180,E1 -21575.715,E2 -21575.715} C_VEL
LIN {X 0,Y 214.482,Z 646.052,A -85,B 0,C 180,E1 -21578.872,E2 -21578.872} C_VEL
LIN {X 0,Y 219.572,Z 637.964,A -85,B 0,C 180,E1 -21582.091,E2 -21582.091} C_VEL
LIN {X 0,Y 225.317,Z 628.062,A -85,B 0,C 180,E1 -21585.225,E2 -21585.225} C_VEL
LIN {X 0,Y 231.154,Z 617.17,A -85,B 0,C 180,E1 -21587.934,E2 -21587.934} C_VEL
LIN {X 0,Y 236.938,Z 604.991,A -85,B 0,C 180,E1 -21590.342,E2 -21590.342} C_VEL
LIN {X 0,Y 238.922,Z 600.417,A -85,B 0,C 180,E1 -21591.115,E2 -21591.115} C_VEL
LIN {X 0,Y 239.305,Z 598.511,A -85,B 0,C 180,E1 -21591.555,E2 -21591.555} C_VEL
LIN {X 0,Y 238.864,Z 591.134,A -85,B 0,C 180,E1 -21593.854,E2 -21593.854} C_VEL
LIN {X 0,Y 237.71,Z 584.417,A -85,B 0,C 180,E1 -21596.185,E2 -21596.185} C_VEL
LIN {X 0,Y 236.348,Z 579.021,A -85,B 0,C 180,E1 -21598.295,E2 -21598.295} C_VEL
LIN {X 0,Y 233.615,Z 571.913,A -85,B 0,C 180,E1 -21601.723,E2 -21601.723} C_VEL
LIN {X 0,Y 232.323,Z 568.789,A -85,B 0,C 180,E1 -21603.468,E2 -21603.468} C_VEL
LIN {X 0,Y 230.86,Z 566.297,A -85,B 0,C 180,E1 -21605.239,E2 -21605.239} C_VEL
LIN {X 0,Y 228.406,Z 562.222,A -85,B 0,C 180,E1 -21608.849,E2 -21608.849} C_VEL
LIN {X 0,Y 226.503,Z 559.48,A -85,B 0,C 180,E1 -21612.544,E2 -21612.544} C_VEL
LIN {X 0,Y 225.852,Z 558.73,A -85,B 0,C 180,E1 -21614.414,E2 -21614.414} C_VEL
LIN {X 0,Y 224.857,Z 558.915,A -85,B 0,C 180,E1 -21618.213,E2 -21618.213} C_VEL
LIN {X 0,Y 224.891,Z 560.013,A -85,B 0,C 180,E1 -21622.024,E2 -21622.024} C_VEL
LIN {X 0,Y 225.928,Z 562.087,A -85,B 0,C 180,E1 -21625.816,E2 -21625.816} C_VEL
LIN {X 0,Y 226.272,Z 562.936,A -85,B 0,C 180,E1 -21626.726,E2 -21626.726} C_VEL
LIN {X 0,Y 227.356,Z 566.977,A -85,B 0,C 180,E1 -21629.642,E2 -21629.642} C_VEL
LIN {X 0,Y 228.602,Z 569.383,A -85,B 0,C 180,E1 -21631.509,E2 -21631.509} C_VEL
LIN {X 0,Y 230.596,Z 575.045,A -85,B 0,C 180,E1 -21634.624,E2 -21634.624} C_VEL
LIN {X 0,Y 232.413,Z 580.85,A -85,B 0,C 180,E1 -21637.213,E2 -21637.213} C_VEL
LIN {X 0,Y 234.263,Z 587.748,A -85,B 0,C 180,E1 -21639.849,E2 -21639.849} C_VEL
LIN {X 0,Y 234.878,Z 595.062,A -85,B 0,C 180,E1 -21641.936,E2 -21641.936} C_VEL
LIN {X 0,Y 234.785,Z 605.212,A -85,B 0,C 180,E1 -21644.536,E2 -21644.536} C_VEL
LIN {X 0,Y 233.801,Z 614.895,A -85,B 0,C 180,E1 -21646.85,E2 -21646.85} C_VEL
LIN {X 0,Y 231.942,Z 624.947,A -85,B 0,C 180,E1 -21649.245,E2 -21649.245} C_VEL
LIN {X 0,Y 231.384,Z 627.233,A -85,B 0,C 180,E1 -21649.787,E2 -21649.787} C_VEL
LIN {X 0,Y 225.811,Z 638.411,A -85,B 0,C 180,E1 -21652.071,E2 -21652.071} C_VEL
LIN {X 0,Y 219.916,Z 649.421,A -85,B 0,C 180,E1 -21654.883,E2 -21654.883} C_VEL
LIN {X 0,Y 217.905,Z 653.006,A -85,B 0,C 180,E1 -21655.953,E2 -21655.953} C_VEL
LIN {X 0,Y 215.326,Z 656.601,A -85,B 0,C 180,E1 -21657.002,E2 -21657.002} C_VEL
LIN {X 0,Y 209.684,Z 662.173,A -85,B 0,C 180,E1 -21658.603,E2 -21658.603} C_VEL
LIN {X 0,Y 204.176,Z 667.311,A -85,B 0,C 180,E1 -21660.373,E2 -21660.373} C_VEL
LIN {X 0,Y 201.857,Z 670.129,A -85,B 0,C 180,E1 -21661.672,E2 -21661.672} C_VEL
LIN {X 0,Y 198.286,Z 675.735,A -85,B 0,C 180,E1 -21664.828,E2 -21664.828} C_VEL
LIN {X 0,Y 194.929,Z 681.317,A -85,B 0,C 180,E1 -21668.866,E2 -21668.866} C_VEL
LIN {X 0,Y 192.474,Z 685.667,A -85,B 0,C 180,E1 -21673.015,E2 -21673.015} C_VEL
LIN {X 0,Y 190.968,Z 688.84,A -85,B 0,C 180,E1 -21677.242,E2 -21677.242} C_VEL
LIN {X 0,Y 190.365,Z 690.892,A -85,B 0,C 180,E1 -21681.507,E2 -21681.507} C_VEL
LIN {X 0,Y 190.431,Z 691.8,A -85,B 0,C 180,E1 -21685.766,E2 -21685.766} C_VEL
LIN {X 0,Y 190.573,Z 691.799,A -85,B 0,C 180,E1 -21687.886,E2 -21687.886} C_VEL
LIN {X 0,Y 190.665,Z 691.5,A -85,B 0,C 180,E1 -21689.999,E2 -21689.999} C_VEL
LIN {X 0,Y 190.551,Z 689.968,A -85,B 0,C 180,E1 -21694.229,E2 -21694.229} C_VEL
LIN {X 0,Y 190.501,Z 688.731,A -85,B 0,C 180,E1 -21696.353,E2 -21696.353} C_VEL
LIN {X 0,Y 190.683,Z 685.282,A -85,B 0,C 180,E1 -21700.618,E2 -21700.618} C_VEL
LIN {X 0,Y 191.625,Z 680.479,A -85,B 0,C 180,E1 -21704.875,E2 -21704.875} C_VEL
LIN {X 0,Y 193.479,Z 674.01,A -85,B 0,C 180,E1 -21709.192,E2 -21709.192} C_VEL
LIN {X 0,Y 196.038,Z 666.252,A -85,B 0,C 180,E1 -21713.224,E2 -21713.224} C_VEL
LIN {X 0,Y 199.259,Z 657.808,A -85,B 0,C 180,E1 -21716.723,E2 -21716.723} C_VEL
LIN {X 0,Y 202.638,Z 648.463,A -85,B 0,C 180,E1 -21719.882,E2 -21719.882} C_VEL
LIN {X 0,Y 206.749,Z 637.183,A -85,B 0,C 180,E1 -21722.947,E2 -21722.947} C_VEL
LIN {X 0,Y 211.065,Z 624.768,A -85,B 0,C 180,E1 -21725.639,E2 -21725.639} C_VEL
LIN {X 0,Y 212.605,Z 620.09,A -85,B 0,C 180,E1 -21726.512,E2 -21726.512} C_VEL
LIN {X 0,Y 212.75,Z 609.672,A -85,B 0,C 180,E1 -21728.654,E2 -21728.654} C_VEL
LIN {X 0,Y 212.106,Z 597.354,A -85,B 0,C 180,E1 -21731.009,E2 -21731.009} C_VEL
LIN {X 0,Y 210.764,Z 584.998,A -85,B 0,C 180,E1 -21733.197,E2 -21733.197} C_VEL
LIN {X 0,Y 208.226,Z 570.741,A -85,B 0,C 180,E1 -21735.546,E2 -21735.546} C_VEL
LIN {X 0,Y 205.212,Z 559.099,A -85,B 0,C 180,E1 -21737.439,E2 -21737.439} C_VEL
LIN {X 0,Y 201.415,Z 549.921,A -85,B 0,C 180,E1 -21739.144,E2 -21739.144} C_VEL
LIN {X 0,Y 198.872,Z 544.863,A -85,B 0,C 180,E1 -21740.157,E2 -21740.157} C_VEL
LIN {X 0,Y 196.458,Z 540.243,A -85,B 0,C 180,E1 -21741.078,E2 -21741.078} C_VEL
LIN {X 0,Y 194.716,Z 537.202,A -85,B 0,C 180,E1 -21741.741,E2 -21741.741} C_VEL
LIN {X 0,Y 194.264,Z 535.324,A -85,B 0,C 180,E1 -21742.048,E2 -21742.048} C_VEL
LIN {X 0,Y 193.662,Z 531.648,A -85,B 0,C 180,E1 -21747.021,E2 -21747.021} C_VEL
LIN {X 0,Y 193.2,Z 528.38,A -85,B 0,C 180,E1 -21751.778,E2 -21751.778} C_VEL
LIN {X 0,Y 192.665,Z 525.112,A -85,B 0,C 180,E1 -21756.913,E2 -21756.913} C_VEL
LIN {X 0,Y 192.725,Z 525.107,A -85,B 0,C 180,E1 -21761.458,E2 -21761.458} C_VEL
LIN {X 0,Y 192.765,Z 525.098,A -85,B 0,C 180,E1 -21765.215,E2 -21765.215} C_VEL
LIN {X 0,Y 192.975,Z 525.049,A -85,B 0,C 180,E1 -21769.509,E2 -21769.509} C_VEL
LIN {X 0,Y 193.062,Z 525.034,A -85,B 0,C 180,E1 -21771.628,E2 -21771.628} C_VEL
LIN {X 0,Y 193.26,Z 525.027,A -85,B 0,C 180,E1 -21777.917,E2 -21777.917} C_VEL
LIN {X 0,Y 193.437,Z 524.983,A -85,B 0,C 180,E1 -21780.001,E2 -21780.001} C_VEL
LIN {X 0,Y 192.972,Z 525.063,A -85,B 0,C 180,E1 -21784.178,E2 -21784.178} C_VEL
LIN {X 0,Y 193.036,Z 525.059,A -85,B 0,C 180,E1 -21788.375,E2 -21788.375} C_VEL
LIN {X 0,Y 192.796,Z 525.055,A -85,B 0,C 180,E1 -21792.635,E2 -21792.635} C_VEL
LIN {X 0,Y 192.765,Z 525.095,A -85,B 0,C 180,E1 -21796.959,E2 -21796.959} C_VEL
LIN {X 0,Y 192.637,Z 525.095,A -85,B 0,C 180,E1 -21801.398,E2 -21801.398} C_VEL
LIN {X 0,Y 192.66,Z 525.072,A -85,B 0,C 180,E1 -21804.226,E2 -21804.226} C_VEL
LIN {X 0,Y 192.646,Z 525.11,A -85,B 0,C 180,E1 -21808.894,E2 -21808.894} C_VEL
LIN {X 0,Y 192.597,Z 525.1,A -85,B 0,C 180,E1 -21813.187,E2 -21813.187} C_VEL
LIN {X 0,Y 192.611,Z 525.103,A -85,B 0,C 180,E1 -21818.339,E2 -21818.339} C_VEL
LIN {X 0,Y 192.631,Z 525.108,A -85,B 0,C 180,E1 -21823.143,E2 -21823.143} C_VEL
LIN {X 0,Y 192.619,Z 525.089,A -85,B 0,C 180,E1 -21826.865,E2 -21826.865} C_VEL
LIN {X 0,Y 192.612,Z 525.121,A -85,B 0,C 180,E1 -21831.665,E2 -21831.665} C_VEL
LIN {X 0,Y 192.601,Z 525.104,A -85,B 0,C 180,E1 -21836.817,E2 -21836.817} C_VEL
LIN {X 0,Y 192.666,Z 525.106,A -85,B 0,C 180,E1 -21841.694,E2 -21841.694} C_VEL
LIN {X 0,Y 192.709,Z 525.107,A -85,B 0,C 180,E1 -21846.351,E2 -21846.351} C_VEL
LIN {X 0,Y 192.735,Z 525.092,A -85,B 0,C 180,E1 -21851.459,E2 -21851.459} C_VEL
LIN {X 0,Y 192.775,Z 525.085,A -85,B 0,C 180,E1 -21855.216,E2 -21855.216} C_VEL
LIN {X 0,Y 192.874,Z 525.087,A -85,B 0,C 180,E1 -21858.27,E2 -21858.27} C_VEL
LIN {X 0,Y 193.803,Z 527.783,A -85,B 0,C 180,E1 -21858.754,E2 -21858.754} C_VEL
LIN {X 0,Y 195.698,Z 530.088,A -85,B 0,C 180,E1 -21859.475,E2 -21859.475} C_VEL
LIN {X 0,Y 197.639,Z 533.352,A -85,B 0,C 180,E1 -21860.268,E2 -21860.268} C_VEL
LIN {X 0,Y 204.309,Z 545.341,A -85,B 0,C 180,E1 -21863.147,E2 -21863.147} C_VEL
LIN {X 0,Y 209.599,Z 555.719,A -85,B 0,C 180,E1 -21865.606,E2 -21865.606} C_VEL
LIN {X 0,Y 214.402,Z 569.013,A -85,B 0,C 180,E1 -21868.508,E2 -21868.508} C_VEL
LIN {X 0,Y 216.457,Z 578.255,A -85,B 0,C 180,E1 -21870.466,E2 -21870.466} C_VEL
LIN {X 0,Y 217.768,Z 585.658,A -85,B 0,C 180,E1 -21872.082,E2 -21872.082} C_VEL
LIN {X 0,Y 216.305,Z 591.508,A -85,B 0,C 180,E1 -21873.027,E2 -21873.027} C_VEL
LIN {X 0,Y 212.613,Z 603.459,A -85,B 0,C 180,E1 -21875.194,E2 -21875.194} C_VEL
LIN {X 0,Y 208.751,Z 614.906,A -85,B 0,C 180,E1 -21877.74,E2 -21877.74} C_VEL
LIN {X 0,Y 205.224,Z 624.613,A -85,B 0,C 180,E1 -21880.358,E2 -21880.358} C_VEL
LIN {X 0,Y 201.541,Z 634.322,A -85,B 0,C 180,E1 -21883.556,E2 -21883.556} C_VEL
LIN {X 0,Y 198.359,Z 642.637,A -85,B 0,C 180,E1 -21886.933,E2 -21886.933} C_VEL
LIN {X 0,Y 195.504,Z 650.352,A -85,B 0,C 180,E1 -21890.826,E2 -21890.826} C_VEL
LIN {X 0,Y 193.371,Z 656.404,A -85,B 0,C 180,E1 -21894.683,E2 -21894.683} C_VEL
LIN {X 0,Y 191.915,Z 661.086,A -85,B 0,C 180,E1 -21898.489,E2 -21898.489} C_VEL
LIN {X 0,Y 190.892,Z 664.553,A -85,B 0,C 180,E1 -21902.135,E2 -21902.135} C_VEL
LIN {X 0,Y 190.242,Z 667.28,A -85,B 0,C 180,E1 -21906.234,E2 -21906.234} C_VEL
LIN {X 0,Y 190.107,Z 668.566,A -85,B 0,C 180,E1 -21909.072,E2 -21909.072} C_VEL
LIN {X 0,Y 190.236,Z 669.366,A -85,B 0,C 180,E1 -21912.363,E2 -21912.363} C_VEL
LIN {X 0,Y 190.68,Z 669.529,A -85,B 0,C 180,E1 -21915.548,E2 -21915.548} C_VEL
LIN {X 0,Y 191.875,Z 668.625,A -85,B 0,C 180,E1 -21920.281,E2 -21920.281} C_VEL
LIN {X 0,Y 193.763,Z 666.585,A -85,B 0,C 180,E1 -21924.525,E2 -21924.525} C_VEL
LIN {X 0,Y 196.652,Z 663.014,A -85,B 0,C 180,E1 -21929.062,E2 -21929.062} C_VEL
LIN {X 0,Y 199.896,Z 658.849,A -85,B 0,C 180,E1 -21932.802,E2 -21932.802} C_VEL
LIN {X 0,Y 204.113,Z 653.212,A -85,B 0,C 180,E1 -21936.603,E2 -21936.603} C_VEL
LIN {X 0,Y 209.2,Z 645.892,A -85,B 0,C 180,E1 -21940.369,E2 -21940.369} C_VEL
LIN {X 0,Y 214.247,Z 638.358,A -85,B 0,C 180,E1 -21943.4,E2 -21943.4} C_VEL
LIN {X 0,Y 219.694,Z 629.461,A -85,B 0,C 180,E1 -21946.28,E2 -21946.28} C_VEL
LIN {X 0,Y 225.472,Z 619.291,A -85,B 0,C 180,E1 -21948.894,E2 -21948.894} C_VEL
LIN {X 0,Y 231.298,Z 607.853,A -85,B 0,C 180,E1 -21951.261,E2 -21951.261} C_VEL
LIN {X 0,Y 233.811,Z 602.423,A -85,B 0,C 180,E1 -21952.226,E2 -21952.226} C_VEL
LIN {X 0,Y 233.943,Z 596.917,A -85,B 0,C 180,E1 -21953.964,E2 -21953.964} C_VEL
LIN {X 0,Y 233.336,Z 590.893,A -85,B 0,C 180,E1 -21956.113,E2 -21956.113} C_VEL
LIN {X 0,Y 232.364,Z 585.427,A -85,B 0,C 180,E1 -21958.266,E2 -21958.266} C_VEL
LIN {X 0,Y 230.069,Z 578.399,A -85,B 0,C 180,E1 -21961.75,E2 -21961.75} C_VEL
LIN {X 0,Y 228.359,Z 573.937,A -85,B 0,C 180,E1 -21964.412,E2 -21964.412} C_VEL
LIN {X 0,Y 225.524,Z 568.704,A -85,B 0,C 180,E1 -21968.963,E2 -21968.963} C_VEL
LIN {X 0,Y 223.714,Z 565.855,A -85,B 0,C 180,E1 -21973.127,E2 -21973.127} C_VEL
LIN {X 0,Y 223.261,Z 565.383,A -85,B 0,C 180,E1 -21974.585,E2 -21974.585} C_VEL
LIN {X 0,Y 222.334,Z 565.622,A -85,B 0,C 180,E1 -21978.504,E2 -21978.504} C_VEL
LIN {X 0,Y 222.423,Z 566.802,A -85,B 0,C 180,E1 -21982.282,E2 -21982.282} C_VEL
LIN {X 0,Y 223.439,Z 569.1,A -85,B 0,C 180,E1 -21986.126,E2 -21986.126} C_VEL
LIN {X 0,Y 225.478,Z 575.868,A -85,B 0,C 180,E1 -21991.274,E2 -21991.274} C_VEL
LIN {X 0,Y 227.197,Z 581.699,A -85,B 0,C 180,E1 -21994.508,E2 -21994.508} C_VEL
LIN {X 0,Y 228.875,Z 587.859,A -85,B 0,C 180,E1 -21997.333,E2 -21997.333} C_VEL
LIN {X 0,Y 229.95,Z 593.681,A -85,B 0,C 180,E1 -21999.521,E2 -21999.521} C_VEL
LIN {X 0,Y 230.02,Z 602.019,A -85,B 0,C 180,E1 -22001.92,E2 -22001.92} C_VEL
LIN {X 0,Y 229.401,Z 610.632,A -85,B 0,C 180,E1 -22004.212,E2 -22004.212} C_VEL
LIN {X 0,Y 227.733,Z 620.926,A -85,B 0,C 180,E1 -22006.785,E2 -22006.785} C_VEL
LIN {X 0,Y 225.954,Z 628.202,A -85,B 0,C 180,E1 -22008.613,E2 -22008.613} C_VEL
LIN {X 0,Y 220.282,Z 639.157,A -85,B 0,C 180,E1 -22010.941,E2 -22010.941} C_VEL
LIN {X 0,Y 214.163,Z 649.945,A -85,B 0,C 180,E1 -22013.794,E2 -22013.794} C_VEL
LIN {X 0,Y 208.639,Z 659.027,A -85,B 0,C 180,E1 -22016.812,E2 -22016.812} C_VEL
LIN {X 0,Y 203.892,Z 666.746,A -85,B 0,C 180,E1 -22020.013,E2 -22020.013} C_VEL
LIN {X 0,Y 201.857,Z 670.129,A -85,B 0,C 180,E1 -22021.672,E2 -22021.672} C_VEL
LIN {X 0,Y 199.595,Z 672.845,A -85,B 0,C 180,E1 -22023.033,E2 -22023.033} C_VEL
LIN {X 0,Y 194.382,Z 676.901,A -85,B 0,C 180,E1 -22025.185,E2 -22025.185} C_VEL
LIN {X 0,Y 189.377,Z 680.473,A -85,B 0,C 180,E1 -22027.507,E2 -22027.507} C_VEL
LIN {X 0,Y 187.495,Z 682.359,A -85,B 0,C 180,E1 -22029.107,E2 -22029.107} C_VEL
LIN {X 0,Y 185.625,Z 685.478,A -85,B 0,C 180,E1 -22032.368,E2 -22032.368} C_VEL
LIN {X 0,Y 183.972,Z 688.555,A -85,B 0,C 180,E1 -22036.749,E2 -22036.749} C_VEL
LIN {X 0,Y 183.306,Z 690.519,A -85,B 0,C 180,E1 -22041.177,E2 -22041.177} C_VEL
LIN {X 0,Y 183.354,Z 691.376,A -85,B 0,C 180,E1 -22045.602,E2 -22045.602} C_VEL
LIN {X 0,Y 183.48,Z 691.345,A -85,B 0,C 180,E1 -22047.804,E2 -22047.804} C_VEL
LIN {X 0,Y 183.597,Z 691.009,A -85,B 0,C 180,E1 -22049.999,E2 -22049.999} C_VEL
LIN {X 0,Y 183.54,Z 690.358,A -85,B 0,C 180,E1 -22052.193,E2 -22052.193} C_VEL
LIN {X 0,Y 183.502,Z 688.963,A -85,B 0,C 180,E1 -22055.271,E2 -22055.271} C_VEL
LIN {X 0,Y 183.431,Z 686.507,A -85,B 0,C 180,E1 -22058.814,E2 -22058.814} C_VEL
LIN {X 0,Y 184.051,Z 682.301,A -85,B 0,C 180,E1 -22063.243,E2 -22063.243} C_VEL
LIN {X 0,Y 185.522,Z 676.676,A -85,B 0,C 180,E1 -22067.64,E2 -22067.64} C_VEL
LIN {X 0,Y 187.929,Z 669.487,A -85,B 0,C 180,E1 -22071.959,E2 -22071.959} C_VEL
LIN {X 0,Y 190.84,Z 661.778,A -85,B 0,C 180,E1 -22075.638,E2 -22075.638} C_VEL
LIN {X 0,Y 194.432,Z 652.483,A -85,B 0,C 180,E1 -22079.206,E2 -22079.206} C_VEL
LIN {X 0,Y 198.016,Z 643.019,A -85,B 0,C 180,E1 -22082.164,E2 -22082.164} C_VEL
LIN {X 0,Y 202.578,Z 630.8,A -85,B 0,C 180,E1 -22085.222,E2 -22085.222} C_VEL
LIN {X 0,Y 206.078,Z 620.795,A -85,B 0,C 180,E1 -22087.251,E2 -22087.251} C_VEL
LIN {X 0,Y 206.245,Z 609.3,A -85,B 0,C 180,E1 -22089.74,E2 -22089.74} C_VEL
LIN {X 0,Y 205.72,Z 597.92,A -85,B 0,C 180,E1 -22092.01,E2 -22092.01} C_VEL
LIN {X 0,Y 204.274,Z 584.298,A -85,B 0,C 180,E1 -22094.512,E2 -22094.512} C_VEL
LIN {X 0,Y 202.087,Z 571.778,A -85,B 0,C 180,E1 -22096.688,E2 -22096.688} C_VEL
LIN {X 0,Y 199.278,Z 560.939,A -85,B 0,C 180,E1 -22098.605,E2 -22098.605} C_VEL
LIN {X 0,Y 194.433,Z 549.862,A -85,B 0,C 180,E1 -22100.845,E2 -22100.845} C_VEL
LIN {X 0,Y 191.391,Z 544.117,A -85,B 0,C 180,E1 -22102.141,E2 -22102.141} C_VEL
LIN {X 0,Y 189.15,Z 539.647,A -85,B 0,C 180,E1 -22103.097,E2 -22103.097} C_VEL
LIN {X 0,Y 187.422,Z 536.68,A -85,B 0,C 180,E1 -22103.801,E2 -22103.801} C_VEL
LIN {X 0,Y 186.955,Z 534.808,A -85,B 0,C 180,E1 -22104.113,E2 -22104.113} C_VEL
LIN {X 0,Y 186.506,Z 532.02,A -85,B 0,C 180,E1 -22108.16,E2 -22108.16} C_VEL
LIN {X 0,Y 186.322,Z 530.32,A -85,B 0,C 180,E1 -22110.637,E2 -22110.637} C_VEL
LIN {X 0,Y 185.853,Z 527.315,A -85,B 0,C 180,E1 -22115.421,E2 -22115.421} C_VEL
LIN {X 0,Y 185.612,Z 525.993,A -85,B 0,C 180,E1 -22117.751,E2 -22117.751} C_VEL
LIN {X 0,Y 185.683,Z 525.982,A -85,B 0,C 180,E1 -22122.375,E2 -22122.375} C_VEL
LIN {X 0,Y 185.758,Z 525.971,A -85,B 0,C 180,E1 -22126.88,E2 -22126.88} C_VEL
LIN {X 0,Y 186.007,Z 525.91,A -85,B 0,C 180,E1 -22131.308,E2 -22131.308} C_VEL
LIN {X 0,Y 186.204,Z 525.906,A -85,B 0,C 180,E1 -22137.838,E2 -22137.838} C_VEL
LIN {X 0,Y 186.401,Z 525.858,A -85,B 0,C 180,E1 -22140.001,E2 -22140.001} C_VEL
LIN {X 0,Y 185.918,Z 525.943,A -85,B 0,C 180,E1 -22144.337,E2 -22144.337} C_VEL
LIN {X 0,Y 185.981,Z 525.934,A -85,B 0,C 180,E1 -22148.695,E2 -22148.695} C_VEL
LIN {X 0,Y 185.723,Z 525.937,A -85,B 0,C 180,E1 -22153.124,E2 -22153.124} C_VEL
LIN {X 0,Y 185.712,Z 525.977,A -85,B 0,C 180,E1 -22157.624,E2 -22157.624} C_VEL
LIN {X 0,Y 185.595,Z 525.961,A -85,B 0,C 180,E1 -22162.253,E2 -22162.253} C_VEL
LIN {X 0,Y 185.558,Z 525.982,A -85,B 0,C 180,E1 -22167.034,E2 -22167.034} C_VEL
LIN {X 0,Y 185.576,Z 525.994,A -85,B 0,C 180,E1 -22169.495,E2 -22169.495} C_VEL
LIN {X 0,Y 185.518,Z 525.966,A -85,B 0,C 180,E1 -22174.629,E2 -22174.629} C_VEL
LIN {X 0,Y 185.566,Z 525.968,A -85,B 0,C 180,E1 -22177.316,E2 -22177.316} C_VEL
LIN {X 0,Y 185.583,Z 525.993,A -85,B 0,C 180,E1 -22180.768,E2 -22180.768} C_VEL
LIN {X 0,Y 185.581,Z 525.962,A -85,B 0,C 180,E1 -22186.018,E2 -22186.018} C_VEL
LIN {X 0,Y 185.56,Z 525.996,A -85,B 0,C 180,E1 -22189.921,E2 -22189.921} C_VEL
LIN {X 0,Y 185.575,Z 525.993,A -85,B 0,C 180,E1 -22192.706,E2 -22192.706} C_VEL
LIN {X 0,Y 185.546,Z 525.993,A -85,B 0,C 180,E1 -22197.977,E2 -22197.977} C_VEL
LIN {X 0,Y 185.583,Z 525.997,A -85,B 0,C 180,E1 -22200.578,E2 -22200.578} C_VEL
LIN {X 0,Y 185.59,Z 525.985,A -85,B 0,C 180,E1 -22205.385,E2 -22205.385} C_VEL
LIN {X 0,Y 185.61,Z 525.973,A -85,B 0,C 180,E1 -22210.077,E2 -22210.077} C_VEL
LIN {X 0,Y 185.704,Z 525.968,A -85,B 0,C 180,E1 -22214.639,E2 -22214.639} C_VEL
LIN {X 0,Y 185.718,Z 525.964,A -85,B 0,C 180,E1 -22216.251,E2 -22216.251} C_VEL
LIN {X 0,Y 186.748,Z 528.81,A -85,B 0,C 180,E1 -22216.848,E2 -22216.848} C_VEL
LIN {X 0,Y 188.607,Z 531.11,A -85,B 0,C 180,E1 -22217.606,E2 -22217.606} C_VEL
LIN {X 0,Y 190.778,Z 534.572,A -85,B 0,C 180,E1 -22218.534,E2 -22218.534} C_VEL
LIN {X 0,Y 195.124,Z 541.856,A -85,B 0,C 180,E1 -22220.501,E2 -22220.501} C_VEL
LIN {X 0,Y 202.37,Z 555.768,A -85,B 0,C 180,E1 -22224.021,E2 -22224.021} C_VEL
LIN {X 0,Y 204.857,Z 561.654,A -85,B 0,C 180,E1 -22225.445,E2 -22225.445} C_VEL
LIN {X 0,Y 209.105,Z 574.442,A -85,B 0,C 180,E1 -22228.416,E2 -22228.416} C_VEL
LIN {X 0,Y 211.268,Z 586.584,A -85,B 0,C 180,E1 -22231.131,E2 -22231.131} C_VEL
LIN {X 0,Y 211.421,Z 587.765,A -85,B 0,C 180,E1 -22231.4,E2 -22231.4} C_VEL
LIN {X 0,Y 207.435,Z 600.635,A -85,B 0,C 180,E1 -22233.643,E2 -22233.643} C_VEL
LIN {X 0,Y 203.399,Z 612.457,A -85,B 0,C 180,E1 -22236.2,E2 -22236.2} C_VEL
LIN {X 0,Y 199.303,Z 623.426,A -85,B 0,C 180,E1 -22239.113,E2 -22239.113} C_VEL
LIN {X 0,Y 195.313,Z 633.625,A -85,B 0,C 180,E1 -22242.469,E2 -22242.469} C_VEL
LIN {X 0,Y 191.982,Z 641.984,A -85,B 0,C 180,E1 -22245.871,E2 -22245.871} C_VEL
LIN {X 0,Y 189.112,Z 649.308,A -85,B 0,C 180,E1 -22249.541,E2 -22249.541} C_VEL
LIN {X 0,Y 186.92,Z 655.298,A -85,B 0,C 180,E1 -22253.254,E2 -22253.254} C_VEL
LIN {X 0,Y 185.294,Z 660.163,A -85,B 0,C 180,E1 -22257.075,E2 -22257.075} C_VEL
LIN {X 0,Y 184.031,Z 664.064,A -85,B 0,C 180,E1 -22261.035,E2 -22261.035} C_VEL
LIN {X 0,Y 183.253,Z 667.023,A -85,B 0,C 180,E1 -22265.119,E2 -22265.119} C_VEL
LIN {X 0,Y 183.022,Z 669.157,A -85,B 0,C 180,E1 -22269.824,E2 -22269.824} C_VEL
LIN {X 0,Y 183.284,Z 669.921,A -85,B 0,C 180,E1 -22273.647,E2 -22273.647} C_VEL
LIN {X 0,Y 183.788,Z 669.971,A -85,B 0,C 180,E1 -22276.599,E2 -22276.599} C_VEL
LIN {X 0,Y 184.577,Z 669.483,A -85,B 0,C 180,E1 -22279.661,E2 -22279.661} C_VEL
LIN {X 0,Y 185.751,Z 668.41,A -85,B 0,C 180,E1 -22282.743,E2 -22282.743} C_VEL
LIN {X 0,Y 188.174,Z 665.862,A -85,B 0,C 180,E1 -22287.21,E2 -22287.21} C_VEL
LIN {X 0,Y 191.6,Z 661.911,A -85,B 0,C 180,E1 -22291.683,E2 -22291.683} C_VEL
LIN {X 0,Y 195.713,Z 656.868,A -85,B 0,C 180,E1 -22295.767,E2 -22295.767} C_VEL
LIN {X 0,Y 200.385,Z 650.836,A -85,B 0,C 180,E1 -22299.467,E2 -22299.467} C_VEL
LIN {X 0,Y 205.806,Z 643.417,A -85,B 0,C 180,E1 -22302.972,E2 -22302.972} C_VEL
LIN {X 0,Y 211.508,Z 635.027,A -85,B 0,C 180,E1 -22306.079,E2 -22306.079} C_VEL
LIN {X 0,Y 217.312,Z 625.793,A -85,B 0,C 180,E1 -22308.81,E2 -22308.81} C_VEL
LIN {X 0,Y 223.539,Z 614.856,A -85,B 0,C 180,E1 -22311.401,E2 -22311.401} C_VEL
LIN {X 0,Y 228.499,Z 605.162,A -85,B 0,C 180,E1 -22313.265,E2 -22313.265} C_VEL
LIN {X 0,Y 228.829,Z 600.784,A -85,B 0,C 180,E1 -22314.713,E2 -22314.713} C_VEL
LIN {X 0,Y 228.41,Z 594.496,A -85,B 0,C 180,E1 -22317.133,E2 -22317.133} C_VEL
LIN {X 0,Y 227.73,Z 589.818,A -85,B 0,C 180,E1 -22319.115,E2 -22319.115} C_VEL
LIN {X 0,Y 225.694,Z 582.59,A -85,B 0,C 180,E1 -22323.001,E2 -22323.001} C_VEL
LIN {X 0,Y 224.318,Z 579.073,A -85,B 0,C 180,E1 -22325.393,E2 -22325.393} C_VEL
LIN {X 0,Y 222.405,Z 575.08,A -85,B 0,C 180,E1 -22329.09,E2 -22329.09} C_VEL
LIN {X 0,Y 220.983,Z 572.491,A -85,B 0,C 180,E1 -22332.862,E2 -22332.862} C_VEL
LIN {X 0,Y 220.413,Z 571.913,A -85,B 0,C 180,E1 -22334.778,E2 -22334.778} C_VEL
LIN {X 0,Y 219.568,Z 572.204,A -85,B 0,C 180,E1 -22338.667,E2 -22338.667} C_VEL
LIN {X 0,Y 219.697,Z 573.489,A -85,B 0,C 180,E1 -22342.573,E2 -22342.573} C_VEL
LIN {X 0,Y 220.144,Z 574.56,A -85,B 0,C 180,E1 -22344.52,E2 -22344.52} C_VEL
LIN {X 0,Y 220.603,Z 576.892,A -85,B 0,C 180,E1 -22346.871,E2 -22346.871} C_VEL
LIN {X 0,Y 221.876,Z 581.297,A -85,B 0,C 180,E1 -22350.451,E2 -22350.451} C_VEL
LIN {X 0,Y 223.206,Z 586.424,A -85,B 0,C 180,E1 -22353.531,E2 -22353.531} C_VEL
LIN {X 0,Y 224.566,Z 592.493,A -85,B 0,C 180,E1 -22356.485,E2 -22356.485} C_VEL
LIN {X 0,Y 225.348,Z 597.683,A -85,B 0,C 180,E1 -22358.59,E2 -22358.59} C_VEL
LIN {X 0,Y 225.08,Z 605.487,A -85,B 0,C 180,E1 -22360.973,E2 -22360.973} C_VEL
LIN {X 0,Y 223.965,Z 615.122,A -85,B 0,C 180,E1 -22363.658,E2 -22363.658} C_VEL
LIN {X 0,Y 221.622,Z 625.689,A -85,B 0,C 180,E1 -22366.449,E2 -22366.449} C_VEL
LIN {X 0,Y 220.371,Z 629.906,A -85,B 0,C 180,E1 -22367.564,E2 -22367.564} C_VEL
LIN {X 0,Y 214.847,Z 639.873,A -85,B 0,C 180,E1 -22369.755,E2 -22369.755} C_VEL
LIN {X 0,Y 208.484,Z 650.454,A -85,B 0,C 180,E1 -22372.643,E2 -22372.643} C_VEL
LIN {X 0,Y 201.964,Z 660.549,A -85,B 0,C 180,E1 -22376.167,E2 -22376.167} C_VEL
LIN {X 0,Y 196.501,Z 668.884,A -85,B 0,C 180,E1 -22379.952,E2 -22379.952} C_VEL
LIN {X 0,Y 191.809,Z 675.746,A -85,B 0,C 180,E1 -22383.915,E2 -22383.915} C_VEL
LIN {X 0,Y 188.249,Z 681.252,A -85,B 0,C 180,E1 -22388.078,E2 -22388.078} C_VEL
LIN {X 0,Y 187.495,Z 682.359,A -85,B 0,C 180,E1 -22389.107,E2 -22389.107} C_VEL
LIN {X 0,Y 185.753,Z 684.106,A -85,B 0,C 180,E1 -22390.76,E2 -22390.76} C_VEL
LIN {X 0,Y 181.486,Z 686.484,A -85,B 0,C 180,E1 -22393.457,E2 -22393.457} C_VEL
LIN {X 0,Y 178.246,Z 687.997,A -85,B 0,C 180,E1 -22395.719,E2 -22395.719} C_VEL
LIN {X 0,Y 176.757,Z 688.949,A -85,B 0,C 180,E1 -22397.54,E2 -22397.54} C_VEL
LIN {X 0,Y 176.559,Z 689.187,A -85,B 0,C 180,E1 -22398.169,E2 -22398.169} C_VEL
LIN {X 0,Y 176.2,Z 690.673,A -85,B 0,C 180,E1 -22403.126,E2 -22403.126} C_VEL
LIN {X 0,Y 176.299,Z 690.921,A -85,B 0,C 180,E1 -22405.426,E2 -22405.426} C_VEL
LIN {X 0,Y 176.53,Z 690.51,A -85,B 0,C 180,E1 -22409.999,E2 -22409.999} C_VEL
LIN {X 0,Y 176.451,Z 689.815,A -85,B 0,C 180,E1 -22412.281,E2 -22412.281} C_VEL
LIN {X 0,Y 176.415,Z 688.527,A -85,B 0,C 180,E1 -22415.17,E2 -22415.17} C_VEL
LIN {X 0,Y 176.372,Z 685.832,A -85,B 0,C 180,E1 -22419.17,E2 -22419.17} C_VEL
LIN {X 0,Y 177.074,Z 681.533,A -85,B 0,C 180,E1 -22423.775,E2 -22423.775} C_VEL
LIN {X 0,Y 178.696,Z 675.81,A -85,B 0,C 180,E1 -22428.337,E2 -22428.337} C_VEL
LIN {X 0,Y 181.258,Z 668.512,A -85,B 0,C 180,E1 -22432.812,E2 -22432.812} C_VEL
LIN {X 0,Y 184.392,Z 660.691,A -85,B 0,C 180,E1 -22436.604,E2 -22436.604} C_VEL
LIN {X 0,Y 188.118,Z 651.246,A -85,B 0,C 180,E1 -22440.287,E2 -22440.287} C_VEL
LIN {X 0,Y 191.957,Z 641.656,A -85,B 0,C 180,E1 -22443.309,E2 -22443.309} C_VEL
LIN {X 0,Y 196.333,Z 630.303,A -85,B 0,C 180,E1 -22446.2,E2 -22446.2} C_VEL
LIN {X 0,Y 199.545,Z 621.465,A -85,B 0,C 180,E1 -22448.048,E2 -22448.048} C_VEL
LIN {X 0,Y 199.809,Z 610.237,A -85,B 0,C 180,E1 -22450.593,E2 -22450.593} C_VEL
LIN {X 0,Y 199.227,Z 596.495,A -85,B 0,C 180,E1 -22453.435,E2 -22453.435} C_VEL
LIN {X 0,Y 197.783,Z 583.213,A -85,B 0,C 180,E1 -22455.995,E2 -22455.995} C_VEL
LIN {X 0,Y 195.797,Z 572.001,A -85,B 0,C 180,E1 -22458.047,E2 -22458.047} C_VEL
LIN {X 0,Y 193.693,Z 564.065,A -85,B 0,C 180,E1 -22459.546,E2 -22459.546} C_VEL
LIN {X 0,Y 189.586,Z 554.216,A -85,B 0,C 180,E1 -22461.702,E2 -22461.702} C_VEL
LIN {X 0,Y 184.522,Z 544.172,A -85,B 0,C 180,E1 -22464.071,E2 -22464.071} C_VEL
LIN {X 0,Y 182.544,Z 540.196,A -85,B 0,C 180,E1 -22464.972,E2 -22464.972} C_VEL
LIN {X 0,Y 180.214,Z 536.273,A -85,B 0,C 180,E1 -22466.012,E2 -22466.012} C_VEL
LIN {X 0,Y 179.658,Z 534.277,A -85,B 0,C 180,E1 -22466.435,E2 -22466.435} C_VEL
LIN {X 0,Y 179.377,Z 532.199,A -85,B 0,C 180,E1 -22469.534,E2 -22469.534} C_VEL
LIN {X 0,Y 178.932,Z 529.08,A -85,B 0,C 180,E1 -22474.601,E2 -22474.601} C_VEL
LIN {X 0,Y 178.539,Z 526.873,A -85,B 0,C 180,E1 -22478.648,E2 -22478.648} C_VEL
LIN {X 0,Y 178.643,Z 526.862,A -85,B 0,C 180,E1 -22481.656,E2 -22481.656} C_VEL
LIN {X 0,Y 178.681,Z 526.853,A -85,B 0,C 180,E1 -22486.35,E2 -22486.35} C_VEL
LIN {X 0,Y 178.935,Z 526.789,A -85,B 0,C 180,E1 -22490.962,E2 -22490.962} C_VEL
LIN {X 0,Y 179.15,Z 526.784,A -85,B 0,C 180,E1 -22497.753,E2 -22497.753} C_VEL
LIN {X 0,Y 179.364,Z 526.732,A -85,B 0,C 180,E1 -22500.001,E2 -22500.001} C_VEL
LIN {X 0,Y 178.866,Z 526.822,A -85,B 0,C 180,E1 -22504.508,E2 -22504.508} C_VEL
LIN {X 0,Y 178.909,Z 526.81,A -85,B 0,C 180,E1 -22509.041,E2 -22509.041} C_VEL
LIN {X 0,Y 178.652,Z 526.82,A -85,B 0,C 180,E1 -22513.654,E2 -22513.654} C_VEL
LIN {X 0,Y 178.634,Z 526.856,A -85,B 0,C 180,E1 -22519.232,E2 -22519.232} C_VEL
LIN {X 0,Y 178.521,Z 526.833,A -85,B 0,C 180,E1 -22525.119,E2 -22525.119} C_VEL
LIN {X 0,Y 178.497,Z 526.875,A -85,B 0,C 180,E1 -22530.788,E2 -22530.788} C_VEL
LIN {X 0,Y 178.482,Z 526.844,A -85,B 0,C 180,E1 -22534.221,E2 -22534.221} C_VEL
LIN {X 0,Y 178.485,Z 526.869,A -85,B 0,C 180,E1 -22539.053,E2 -22539.053} C_VEL
LIN {X 0,Y 178.515,Z 526.872,A -85,B 0,C 180,E1 -22542.013,E2 -22542.013} C_VEL
LIN {X 0,Y 178.527,Z 526.843,A -85,B 0,C 180,E1 -22545.122,E2 -22545.122} C_VEL
LIN {X 0,Y 178.511,Z 526.858,A -85,B 0,C 180,E1 -22548.422,E2 -22548.422} C_VEL
LIN {X 0,Y 178.468,Z 526.867,A -85,B 0,C 180,E1 -22553.796,E2 -22553.796} C_VEL
LIN {X 0,Y 178.492,Z 526.857,A -85,B 0,C 180,E1 -22556.55,E2 -22556.55} C_VEL
LIN {X 0,Y 178.524,Z 526.878,A -85,B 0,C 180,E1 -22560.008,E2 -22560.008} C_VEL
LIN {X 0,Y 178.536,Z 526.857,A -85,B 0,C 180,E1 -22564.878,E2 -22564.878} C_VEL
LIN {X 0,Y 178.626,Z 526.843,A -85,B 0,C 180,E1 -22570.785,E2 -22570.785} C_VEL
LIN {X 0,Y 178.653,Z 526.85,A -85,B 0,C 180,E1 -22574.083,E2 -22574.083} C_VEL
LIN {X 0,Y 179.605,Z 529.576,A -85,B 0,C 180,E1 -22574.686,E2 -22574.686} C_VEL
LIN {X 0,Y 181.603,Z 532.133,A -85,B 0,C 180,E1 -22575.597,E2 -22575.597} C_VEL
LIN {X 0,Y 183.803,Z 535.628,A -85,B 0,C 180,E1 -22576.637,E2 -22576.637} C_VEL
LIN {X 0,Y 188.74,Z 543.625,A -85,B 0,C 180,E1 -22578.997,E2 -22578.997} C_VEL
LIN {X 0,Y 195.597,Z 557.035,A -85,B 0,C 180,E1 -22582.624,E2 -22582.624} C_VEL
LIN {X 0,Y 198.997,Z 564.494,A -85,B 0,C 180,E1 -22584.584,E2 -22584.584} C_VEL
LIN {X 0,Y 202.903,Z 576.599,A -85,B 0,C 180,E1 -22587.563,E2 -22587.563} C_VEL
LIN {X 0,Y 204.87,Z 588.057,A -85,B 0,C 180,E1 -22590.271,E2 -22590.271} C_VEL
LIN {X 0,Y 205.041,Z 589.183,A -85,B 0,C 180,E1 -22590.541,E2 -22590.541} C_VEL
LIN {X 0,Y 200.663,Z 602.747,A -85,B 0,C 180,E1 -22593.012,E2 -22593.012} C_VEL
LIN {X 0,Y 196.228,Z 615.087,A -85,B 0,C 180,E1 -22595.842,E2 -22595.842} C_VEL
LIN {X 0,Y 191.713,Z 626.579,A -85,B 0,C 180,E1 -22599.138,E2 -22599.138} C_VEL
LIN {X 0,Y 188.002,Z 635.667,A -85,B 0,C 180,E1 -22602.361,E2 -22602.361} C_VEL
LIN {X 0,Y 184.395,Z 644.419,A -85,B 0,C 180,E1 -22606.211,E2 -22606.211} C_VEL
LIN {X 0,Y 181.374,Z 651.996,A -85,B 0,C 180,E1 -22610.411,E2 -22610.411} C_VEL
LIN {X 0,Y 179.305,Z 657.356,A -85,B 0,C 180,E1 -22614.157,E2 -22614.157} C_VEL
LIN {X 0,Y 177.719,Z 662.086,A -85,B 0,C 180,E1 -22618.331,E2 -22618.331} C_VEL
LIN {X 0,Y 176.439,Z 666.18,A -85,B 0,C 180,E1 -22623.228,E2 -22623.228} C_VEL
LIN {X 0,Y 175.999,Z 668.387,A -85,B 0,C 180,E1 -22626.998,E2 -22626.998} C_VEL
LIN {X 0,Y 175.968,Z 669.725,A -85,B 0,C 180,E1 -22630.636,E2 -22630.636} C_VEL
LIN {X 0,Y 176.531,Z 670.45,A -85,B 0,C 180,E1 -22635.776,E2 -22635.776} C_VEL
LIN {X 0,Y 177.827,Z 669.831,A -85,B 0,C 180,E1 -22640.775,E2 -22640.775} C_VEL
LIN {X 0,Y 179.795,Z 668.185,A -85,B 0,C 180,E1 -22645.172,E2 -22645.172} C_VEL
LIN {X 0,Y 182.998,Z 664.965,A -85,B 0,C 180,E1 -22650.048,E2 -22650.048} C_VEL
LIN {X 0,Y 186.946,Z 660.631,A -85,B 0,C 180,E1 -22654.456,E2 -22654.456} C_VEL
LIN {X 0,Y 191.618,Z 655.205,A -85,B 0,C 180,E1 -22658.482,E2 -22658.482} C_VEL
LIN {X 0,Y 196.909,Z 648.61,A -85,B 0,C 180,E1 -22662.212,E2 -22662.212} C_VEL
LIN {X 0,Y 203.613,Z 639.769,A -85,B 0,C 180,E1 -22666.017,E2 -22666.017} C_VEL
LIN {X 0,Y 209.416,Z 631.309,A -85,B 0,C 180,E1 -22668.873,E2 -22668.873} C_VEL
LIN {X 0,Y 216.032,Z 620.824,A -85,B 0,C 180,E1 -22671.659,E2 -22671.659} C_VEL
LIN {X 0,Y 222.311,Z 609.685,A -85,B 0,C 180,E1 -22674.007,E2 -22674.007} C_VEL
LIN {X 0,Y 223.488,Z 607.099,A -85,B 0,C 180,E1 -22674.586,E2 -22674.586} C_VEL
LIN {X 0,Y 223.701,Z 601.187,A -85,B 0,C 180,E1 -22676.848,E2 -22676.848} C_VEL
LIN {X 0,Y 223.338,Z 596.012,A -85,B 0,C 180,E1 -22679.098,E2 -22679.098} C_VEL
LIN {X 0,Y 222.034,Z 589.856,A -85,B 0,C 180,E1 -22682.432,E2 -22682.432} C_VEL
LIN {X 0,Y 221.145,Z 586.463,A -85,B 0,C 180,E1 -22684.556,E2 -22684.556} C_VEL
LIN {X 0,Y 219.066,Z 581.34,A -85,B 0,C 180,E1 -22689.23,E2 -22689.23} C_VEL
LIN {X 0,Y 217.857,Z 578.841,A -85,B 0,C 180,E1 -22693.05,E2 -22693.05} C_VEL
LIN {X 0,Y 217.298,Z 578.338,A -85,B 0,C 180,E1 -22694.995,E2 -22694.995} C_VEL
LIN {X 0,Y 216.507,Z 578.915,A -85,B 0,C 180,E1 -22699.718,E2 -22699.718} C_VEL
LIN {X 0,Y 216.725,Z 580.111,A -85,B 0,C 180,E1 -22702.9,E2 -22702.9} C_VEL
LIN {X 0,Y 217.274,Z 582.307,A -85,B 0,C 180,E1 -22705.89,E2 -22705.89} C_VEL
LIN {X 0,Y 218.262,Z 587.087,A -85,B 0,C 180,E1 -22709.938,E2 -22709.938} C_VEL
LIN {X 0,Y 219.477,Z 593.182,A -85,B 0,C 180,E1 -22713.637,E2 -22713.637} C_VEL
LIN {X 0,Y 220.326,Z 597.987,A -85,B 0,C 180,E1 -22716.049,E2 -22716.049} C_VEL
LIN {X 0,Y 220.714,Z 602.634,A -85,B 0,C 180,E1 -22717.987,E2 -22717.987} C_VEL
LIN {X 0,Y 219.999,Z 610.174,A -85,B 0,C 180,E1 -22720.376,E2 -22720.376} C_VEL
LIN {X 0,Y 218.626,Z 618.506,A -85,B 0,C 180,E1 -22722.814,E2 -22722.814} C_VEL
LIN {X 0,Y 215.977,Z 628.361,A -85,B 0,C 180,E1 -22725.566,E2 -22725.566} C_VEL
LIN {X 0,Y 214.626,Z 632.081,A -85,B 0,C 180,E1 -22726.555,E2 -22726.555} C_VEL
LIN {X 0,Y 209.513,Z 640.635,A -85,B 0,C 180,E1 -22728.509,E2 -22728.509} C_VEL
LIN {X 0,Y 202.91,Z 650.974,A -85,B 0,C 180,E1 -22731.431,E2 -22731.431} C_VEL
LIN {X 0,Y 196.086,Z 660.864,A -85,B 0,C 180,E1 -22735.008,E2 -22735.008} C_VEL
LIN {X 0,Y 190.347,Z 669.057,A -85,B 0,C 180,E1 -22738.874,E2 -22738.874} C_VEL
LIN {X 0,Y 185.395,Z 675.76,A -85,B 0,C 180,E1 -22742.941,E2 -22742.941} C_VEL
LIN {X 0,Y 181.634,Z 681.156,A -85,B 0,C 180,E1 -22747.236,E2 -22747.236} C_VEL
LIN {X 0,Y 178.803,Z 685.315,A -85,B 0,C 180,E1 -22751.672,E2 -22751.672} C_VEL
LIN {X 0,Y 176.992,Z 688.278,A -85,B 0,C 180,E1 -22756.216,E2 -22756.216} C_VEL
LIN {X 0,Y 176.559,Z 689.187,A -85,B 0,C 180,E1 -22758.169,E2 -22758.169} C_VEL
LIN {X 0,Y 175.656,Z 689.921,A -85,B 0,C 180,E1 -22760.053,E2 -22760.053} C_VEL
LIN {X 0,Y 172.681,Z 690.522,A -85,B 0,C 180,E1 -22763.158,E2 -22763.158} C_VEL
LIN {X 0,Y 170.319,Z 690.548,A -85,B 0,C 180,E1 -22765.717,E2 -22765.717} C_VEL
LIN {X 0,Y 169.373,Z 690.366,A -85,B 0,C 180,E1 -22767.707,E2 -22767.707} C_VEL
LIN {X 0,Y 169.323,Z 690.253,A -85,B 0,C 180,E1 -22768.381,E2 -22768.381} C_VEL
LIN {X 0,Y 169.463,Z 689.994,A -85,B 0,C 180,E1 -22769.999,E2 -22769.999} C_VEL
LIN {X 0,Y 169.342,Z 688.22,A -85,B 0,C 180,E1 -22774.76,E2 -22774.76} C_VEL
LIN {X 0,Y 169.308,Z 685.14,A -85,B 0,C 180,E1 -22779.556,E2 -22779.556} C_VEL
LIN {X 0,Y 170.113,Z 680.739,A -85,B 0,C 180,E1 -22784.351,E2 -22784.351} C_VEL
LIN {X 0,Y 171.905,Z 674.909,A -85,B 0,C 180,E1 -22789.089,E2 -22789.089} C_VEL
LIN {X 0,Y 174.635,Z 667.488,A -85,B 0,C 180,E1 -22793.729,E2 -22793.729} C_VEL
LIN {X 0,Y 177.975,Z 659.537,A -85,B 0,C 180,E1 -22797.643,E2 -22797.643} C_VEL
LIN {X 0,Y 181.743,Z 650.3,A -85,B 0,C 180,E1 -22801.311,E2 -22801.311} C_VEL
LIN {X 0,Y 185.977,Z 640.186,A -85,B 0,C 180,E1 -22804.528,E2 -22804.528} C_VEL
LIN {X 0,Y 190.528,Z 628.62,A -85,B 0,C 180,E1 -22807.489,E2 -22807.489} C_VEL
LIN {X 0,Y 192.918,Z 622.431,A -85,B 0,C 180,E1 -22808.811,E2 -22808.811} C_VEL
LIN {X 0,Y 193.381,Z 612.647,A -85,B 0,C 180,E1 -22811.152,E2 -22811.152} C_VEL
LIN {X 0,Y 193.103,Z 599.717,A -85,B 0,C 180,E1 -22813.999,E2 -22813.999} C_VEL
LIN {X 0,Y 192.142,Z 588.291,A -85,B 0,C 180,E1 -22816.34,E2 -22816.34} C_VEL
LIN {X 0,Y 190.385,Z 576.318,A -85,B 0,C 180,E1 -22818.692,E2 -22818.692} C_VEL
LIN {X 0,Y 188.47,Z 568.076,A -85,B 0,C 180,E1 -22820.345,E2 -22820.345} C_VEL
LIN {X 0,Y 184.296,Z 557.806,A -85,B 0,C 180,E1 -22822.745,E2 -22822.745} C_VEL
LIN {X 0,Y 179.687,Z 548.323,A -85,B 0,C 180,E1 -22825.121,E2 -22825.121} C_VEL
LIN {X 0,Y 177.394,Z 543.726,A -85,B 0,C 180,E1 -22826.314,E2 -22826.314} C_VEL
LIN {X 0,Y 175.504,Z 539.891,A -85,B 0,C 180,E1 -22827.275,E2 -22827.275} C_VEL
LIN {X 0,Y 173.081,Z 536.161,A -85,B 0,C 180,E1 -22828.421,E2 -22828.421} C_VEL
LIN {X 0,Y 172.402,Z 533.746,A -85,B 0,C 180,E1 -22828.874,E2 -22828.874} C_VEL
LIN {X 0,Y 171.964,Z 530.66,A -85,B 0,C 180,E1 -22834.038,E2 -22834.038} C_VEL
LIN {X 0,Y 171.506,Z 527.752,A -85,B 0,C 180,E1 -22839.541,E2 -22839.541} C_VEL
LIN {X 0,Y 171.578,Z 527.739,A -85,B 0,C 180,E1 -22843.339,E2 -22843.339} C_VEL
LIN {X 0,Y 171.802,Z 527.687,A -85,B 0,C 180,E1 -22849.034,E2 -22849.034} C_VEL
LIN {X 0,Y 171.884,Z 527.68,A -85,B 0,C 180,E1 -22852.955,E2 -22852.955} C_VEL
LIN {X 0,Y 172.098,Z 527.663,A -85,B 0,C 180,E1 -22857.66,E2 -22857.66} C_VEL
LIN {X 0,Y 172.327,Z 527.607,A -85,B 0,C 180,E1 -22860.001,E2 -22860.001} C_VEL
LIN {X 0,Y 171.814,Z 527.702,A -85,B 0,C 180,E1 -22864.694,E2 -22864.694} C_VEL
LIN {X 0,Y 171.845,Z 527.685,A -85,B 0,C 180,E1 -22869.416,E2 -22869.416} C_VEL
LIN {X 0,Y 171.573,Z 527.706,A -85,B 0,C 180,E1 -22874.229,E2 -22874.229} C_VEL
LIN {X 0,Y 171.553,Z 527.735,A -85,B 0,C 180,E1 -22879.576,E2 -22879.576} C_VEL
LIN {X 0,Y 171.458,Z 527.716,A -85,B 0,C 180,E1 -22885.613,E2 -22885.613} C_VEL
LIN {X 0,Y 171.455,Z 527.752,A -85,B 0,C 180,E1 -22890.598,E2 -22890.598} C_VEL
LIN {X 0,Y 171.404,Z 527.719,A -85,B 0,C 180,E1 -22895.033,E2 -22895.033} C_VEL
LIN {X 0,Y 171.437,Z 527.743,A -85,B 0,C 180,E1 -22898.843,E2 -22898.843} C_VEL
LIN {X 0,Y 171.452,Z 527.732,A -85,B 0,C 180,E1 -22904.176,E2 -22904.176} C_VEL
LIN {X 0,Y 171.429,Z 527.747,A -85,B 0,C 180,E1 -22909.011,E2 -22909.011} C_VEL
LIN {X 0,Y 171.441,Z 527.757,A -85,B 0,C 180,E1 -22912.057,E2 -22912.057} C_VEL
LIN {X 0,Y 171.429,Z 527.748,A -85,B 0,C 180,E1 -22917.797,E2 -22917.797} C_VEL
LIN {X 0,Y 171.451,Z 527.758,A -85,B 0,C 180,E1 -22920.537,E2 -22920.537} C_VEL
LIN {X 0,Y 171.46,Z 527.748,A -85,B 0,C 180,E1 -22925.804,E2 -22925.804} C_VEL
LIN {X 0,Y 171.62,Z 527.722,A -85,B 0,C 180,E1 -22931.729,E2 -22931.729} C_VEL
LIN {X 0,Y 172.415,Z 530.274,A -85,B 0,C 180,E1 -22932.296,E2 -22932.296} C_VEL
LIN {X 0,Y 174.604,Z 533.063,A -85,B 0,C 180,E1 -22933.375,E2 -22933.375} C_VEL
LIN {X 0,Y 176.741,Z 536.48,A -85,B 0,C 180,E1 -22934.473,E2 -22934.473} C_VEL
LIN {X 0,Y 181.657,Z 544.466,A -85,B 0,C 180,E1 -22937.064,E2 -22937.064} C_VEL
LIN {X 0,Y 185.379,Z 551.129,A -85,B 0,C 180,E1 -22939.074,E2 -22939.074} C_VEL
LIN {X 0,Y 191.75,Z 564.18,A -85,B 0,C 180,E1 -22942.821,E2 -22942.821} C_VEL
LIN {X 0,Y 194.007,Z 570.294,A -85,B 0,C 180,E1 -22944.444,E2 -22944.444} C_VEL
LIN {X 0,Y 197.047,Z 580.271,A -85,B 0,C 180,E1 -22947.062,E2 -22947.062} C_VEL
LIN {X 0,Y 198.631,Z 590.568,A -85,B 0,C 180,E1 -22949.621,E2 -22949.621} C_VEL
LIN {X 0,Y 194.395,Z 603.464,A -85,B 0,C 180,E1 -22952.073,E2 -22952.073} C_VEL
LIN {X 0,Y 189.936,Z 615.427,A -85,B 0,C 180,E1 -22954.889,E2 -22954.889} C_VEL
LIN {X 0,Y 185.479,Z 626.397,A -85,B 0,C 180,E1 -22958.094,E2 -22958.094} C_VEL
LIN {X 0,Y 181.42,Z 635.906,A -85,B 0,C 180,E1 -22961.544,E2 -22961.544} C_VEL
LIN {X 0,Y 177.685,Z 644.617,A -85,B 0,C 180,E1 -22965.486,E2 -22965.486} C_VEL
LIN {X 0,Y 174.38,Z 652.557,A -85,B 0,C 180,E1 -22970.035,E2 -22970.035} C_VEL
LIN {X 0,Y 172.174,Z 658.101,A -85,B 0,C 180,E1 -22974.092,E2 -22974.092} C_VEL
LIN {X 0,Y 170.6,Z 662.609,A -85,B 0,C 180,E1 -22978.279,E2 -22978.279} C_VEL
LIN {X 0,Y 169.439,Z 666.195,A -85,B 0,C 180,E1 -22982.631,E2 -22982.631} C_VEL
LIN {X 0,Y 168.866,Z 669.057,A -85,B 0,C 180,E1 -22987.742,E2 -22987.742} C_VEL
LIN {X 0,Y 168.94,Z 670.341,A -85,B 0,C 180,E1 -22991.73,E2 -22991.73} C_VEL
LIN {X 0,Y 169.325,Z 670.872,A -85,B 0,C 180,E1 -22995.12,E2 -22995.12} C_VEL
LIN {X 0,Y 170.051,Z 670.819,A -85,B 0,C 180,E1 -22998.603,E2 -22998.603} C_VEL
LIN {X 0,Y 171.149,Z 670.183,A -85,B 0,C 180,E1 -23001.977,E2 -23001.977} C_VEL
LIN {X 0,Y 172.669,Z 669.03,A -85,B 0,C 180,E1 -23005.26,E2 -23005.26} C_VEL
LIN {X 0,Y 174.597,Z 667.378,A -85,B 0,C 180,E1 -23008.446,E2 -23008.446} C_VEL
LIN {X 0,Y 178.238,Z 663.872,A -85,B 0,C 180,E1 -23013.019,E2 -23013.019} C_VEL
LIN {X 0,Y 182.811,Z 659.116,A -85,B 0,C 180,E1 -23017.39,E2 -23017.39} C_VEL
LIN {X 0,Y 188.329,Z 652.935,A -85,B 0,C 180,E1 -23021.591,E2 -23021.591} C_VEL
LIN {X 0,Y 194.479,Z 645.595,A -85,B 0,C 180,E1 -23025.346,E2 -23025.346} C_VEL
LIN {X 0,Y 201.216,Z 636.825,A -85,B 0,C 180,E1 -23028.786,E2 -23028.786} C_VEL
LIN {X 0,Y 207.818,Z 627.414,A -85,B 0,C 180,E1 -23031.666,E2 -23031.666} C_VEL
LIN {X 0,Y 214.875,Z 616.207,A -85,B 0,C 180,E1 -23034.368,E2 -23034.368} C_VEL
LIN {X 0,Y 218.055,Z 610.696,A -85,B 0,C 180,E1 -23035.47,E2 -23035.47} C_VEL
LIN {X 0,Y 218.523,Z 608.359,A -85,B 0,C 180,E1 -23036.311,E2 -23036.311} C_VEL
LIN {X 0,Y 218.663,Z 602.063,A -85,B 0,C 180,E1 -23039.078,E2 -23039.078} C_VEL
